FUNCTION "Generador de Fallas" : VOID	// FC 6
VERSION : 0.1
BEGIN
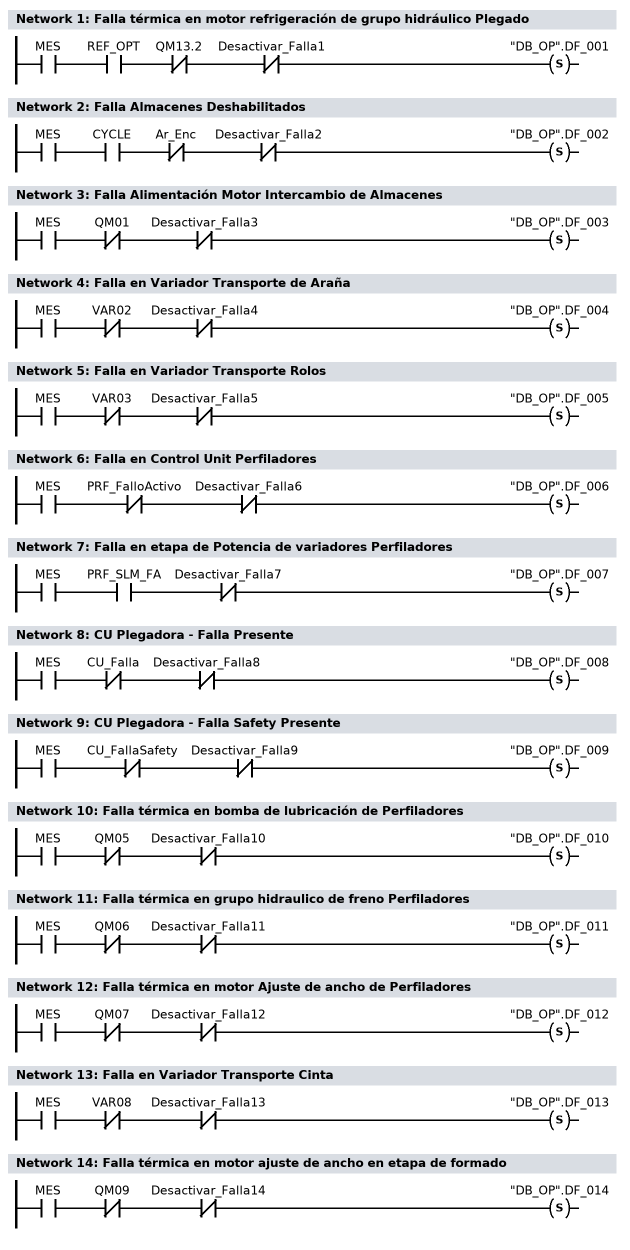
NETWORK
TITLE = Falla térmica en motor refrigeración de grupo hidráulico Plegado
      A     "MES";
      A     "REF_OPT";
      AN    "QM13.2";
      AN    "Desactivar_Falla1";
      S     "DB_OP".DF_001;
NETWORK
TITLE = Falla Almacenes Deshabilitados
      A     "MES";
      A     "CYCLE";
      AN    "Ar_Enc";
      AN    "Desactivar_Falla2";
      S     "DB_OP".DF_002;
NETWORK
TITLE = Falla Alimentación Motor Intercambio de Almacenes
      A     "MES";
      AN    "QM01";
      AN    "Desactivar_Falla3";
      S     "DB_OP".DF_003;
NETWORK
TITLE = Falla en Variador Transporte de Araña
      A     "MES";
      AN    "VAR02";
      AN    "Desactivar_Falla4";
      S     "DB_OP".DF_004;
NETWORK
TITLE = Falla en Variador Transporte Rolos
      A     "MES";
      AN    "VAR03";
      AN    "Desactivar_Falla5";
      S     "DB_OP".DF_005;
NETWORK
TITLE = Falla en Control Unit Perfiladores
      A     "MES";
      AN    "PRF_FalloActivo";
      AN    "Desactivar_Falla6";
      S     "DB_OP".DF_006;
NETWORK
TITLE = Falla en etapa de Potencia de variadores Perfiladores
      A     "MES";
      A     "PRF_SLM_FA";
      AN    "Desactivar_Falla7";
      S     "DB_OP".DF_007;
NETWORK
TITLE = CU Plegadora - Falla Presente
      A     "MES";
      AN    "CU_Falla";
      AN    "Desactivar_Falla8";
      S     "DB_OP".DF_008;
NETWORK
TITLE = CU Plegadora - Falla Safety Presente
      A     "MES";
      AN    "CU_FallaSafety";
      AN    "Desactivar_Falla9";
      S     "DB_OP".DF_009;
NETWORK
TITLE = Falla térmica en bomba de lubricación de Perfiladores
      A     "MES";
      AN    "QM05";
      AN    "Desactivar_Falla10";
      S     "DB_OP".DF_010;
NETWORK
TITLE = Falla térmica en grupo hidraulico de freno Perfiladores
      A     "MES";
      AN    "QM06";
      AN    "Desactivar_Falla11";
      S     "DB_OP".DF_011;
NETWORK
TITLE = Falla térmica en motor Ajuste de ancho de Perfiladores
      A     "MES";
      AN    "QM07";
      AN    "Desactivar_Falla12";
      S     "DB_OP".DF_012;
NETWORK
TITLE = Falla en Variador Transporte Cinta
      A     "MES";
      AN    "VAR08";
      AN    "Desactivar_Falla13";
      S     "DB_OP".DF_013;
NETWORK
TITLE = Falla térmica en motor ajuste de ancho en etapa de formado
      A     "MES";
      AN    "QM09";
      AN    "Desactivar_Falla14";
      S     "DB_OP".DF_014;
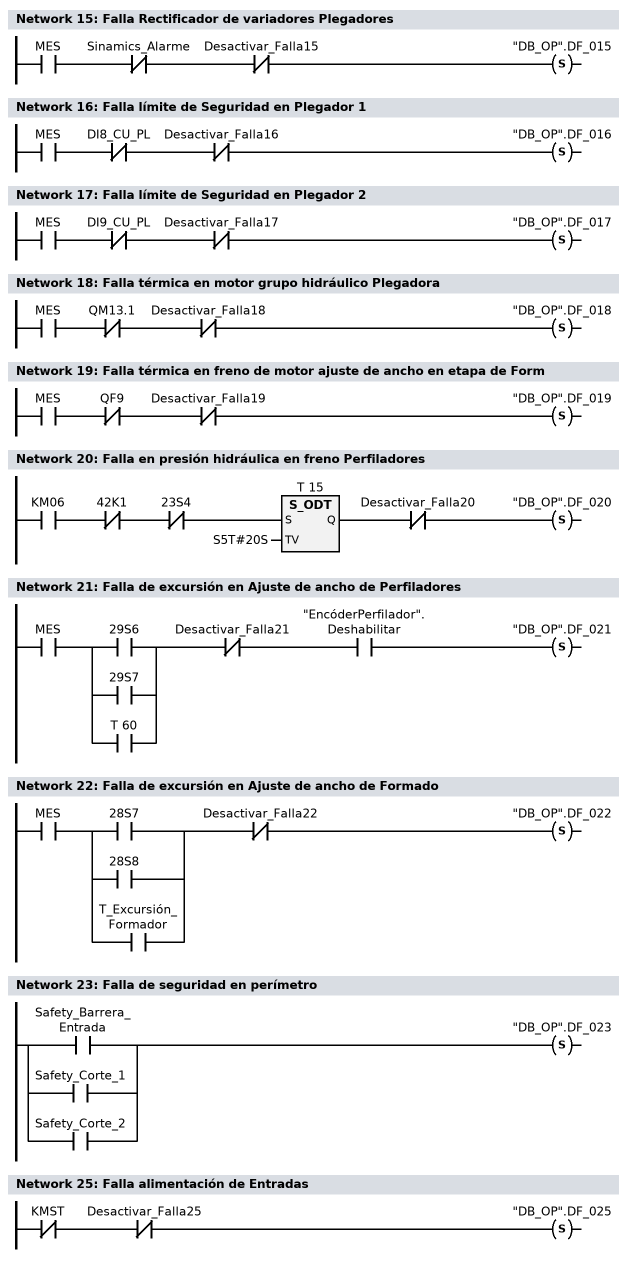
NETWORK
TITLE = Falla Rectificador de variadores Plegadores
      A     "MES";
      AN    "Sinamics_Alarme";
      AN    "Desactivar_Falla15";
      S     "DB_OP".DF_015;
NETWORK
TITLE = Falla límite de Seguridad en Plegador 1
      A     "MES";
      AN    "DI8_CU_PL";
      AN    "Desactivar_Falla16";
      S     "DB_OP".DF_016;
NETWORK
TITLE = Falla límite de Seguridad en Plegador 2
      A     "MES";
      AN    "DI9_CU_PL";
      AN    "Desactivar_Falla17";
      S     "DB_OP".DF_017;
NETWORK
TITLE = Falla térmica en motor grupo hidráulico Plegadora
      A     "MES";
      AN    "QM13.1";
      AN    "Desactivar_Falla18";
      S     "DB_OP".DF_018;
NETWORK
TITLE = Falla térmica en freno de motor ajuste de ancho en etapa de Form
      A     "MES";
      AN    "QF9";
      AN    "Desactivar_Falla19";
      S     "DB_OP".DF_019;
NETWORK
TITLE = Falla en presión hidráulica en freno Perfiladores
      A(;
      A     "KM06";
      AN    "42K1";
      AN    "23S4";
      L     S5T#20S;
      SD    T 15;
      NOP   0;
      NOP   0;
      NOP   0;
      A     T 15;
      );
      AN    "Desactivar_Falla20";
      S     "DB_OP".DF_020;
NETWORK
TITLE = Falla de excursión en Ajuste de ancho de Perfiladores
      A     "MES";
      A(;
      O     "29S6";
      O     "29S7";
      O     T 60;
      );
      AN    "Desactivar_Falla21";
      A     "EncóderPerfilador".Deshabilitar;
      S     "DB_OP".DF_021;
NETWORK
TITLE = Falla de excursión en Ajuste de ancho de Formado
      A     "MES";
      A(;
      O     "28S7";
      O     "28S8";
      O     "T_Excursión_Formador";
      );
      AN    "Desactivar_Falla22";
      S     "DB_OP".DF_022;
NETWORK
TITLE = Falla de seguridad en perímetro
      O     "Safety_Barrera_Entrada";
      O     "Safety_Corte_1";
      O     "Safety_Corte_2";
      S     "DB_OP".DF_023;
NETWORK
TITLE = Reserva
NETWORK
TITLE = Falla alimentación de Entradas
      AN    "KMST";
      AN    "Desactivar_Falla25";
      S     "DB_OP".DF_025;
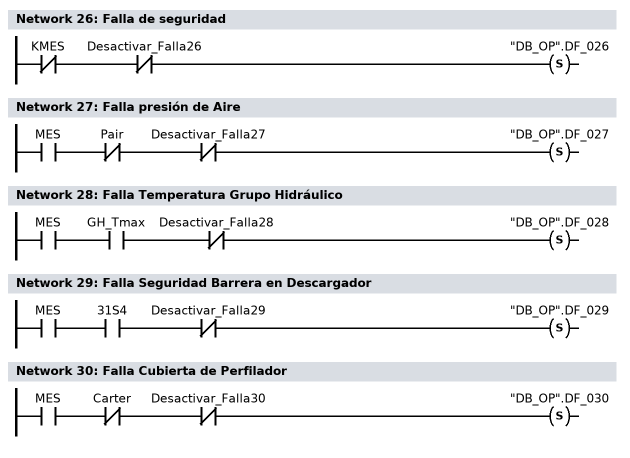
NETWORK
TITLE = Falla de seguridad
      AN    "KMES";
      AN    "Desactivar_Falla26";
      S     "DB_OP".DF_026;
NETWORK
TITLE = Falla presión de Aire
      A     "MES";
      AN    "Pair";
      AN    "Desactivar_Falla27";
      S     "DB_OP".DF_027;
NETWORK
TITLE = Falla Temperatura Grupo Hidráulico
      A     "MES";
      A     "GH_Tmax";
      AN    "Desactivar_Falla28";
      S     "DB_OP".DF_028;
NETWORK
TITLE = Falla Seguridad Barrera en Descargador
      A     "MES";
      A     "31S4";
      AN    "Desactivar_Falla29";
      S     "DB_OP".DF_029;
NETWORK
TITLE = Falla Cubierta de Perfilador
      A     "MES";
      AN    "Carter";
      AN    "Desactivar_Falla30";
      S     "DB_OP".DF_030;
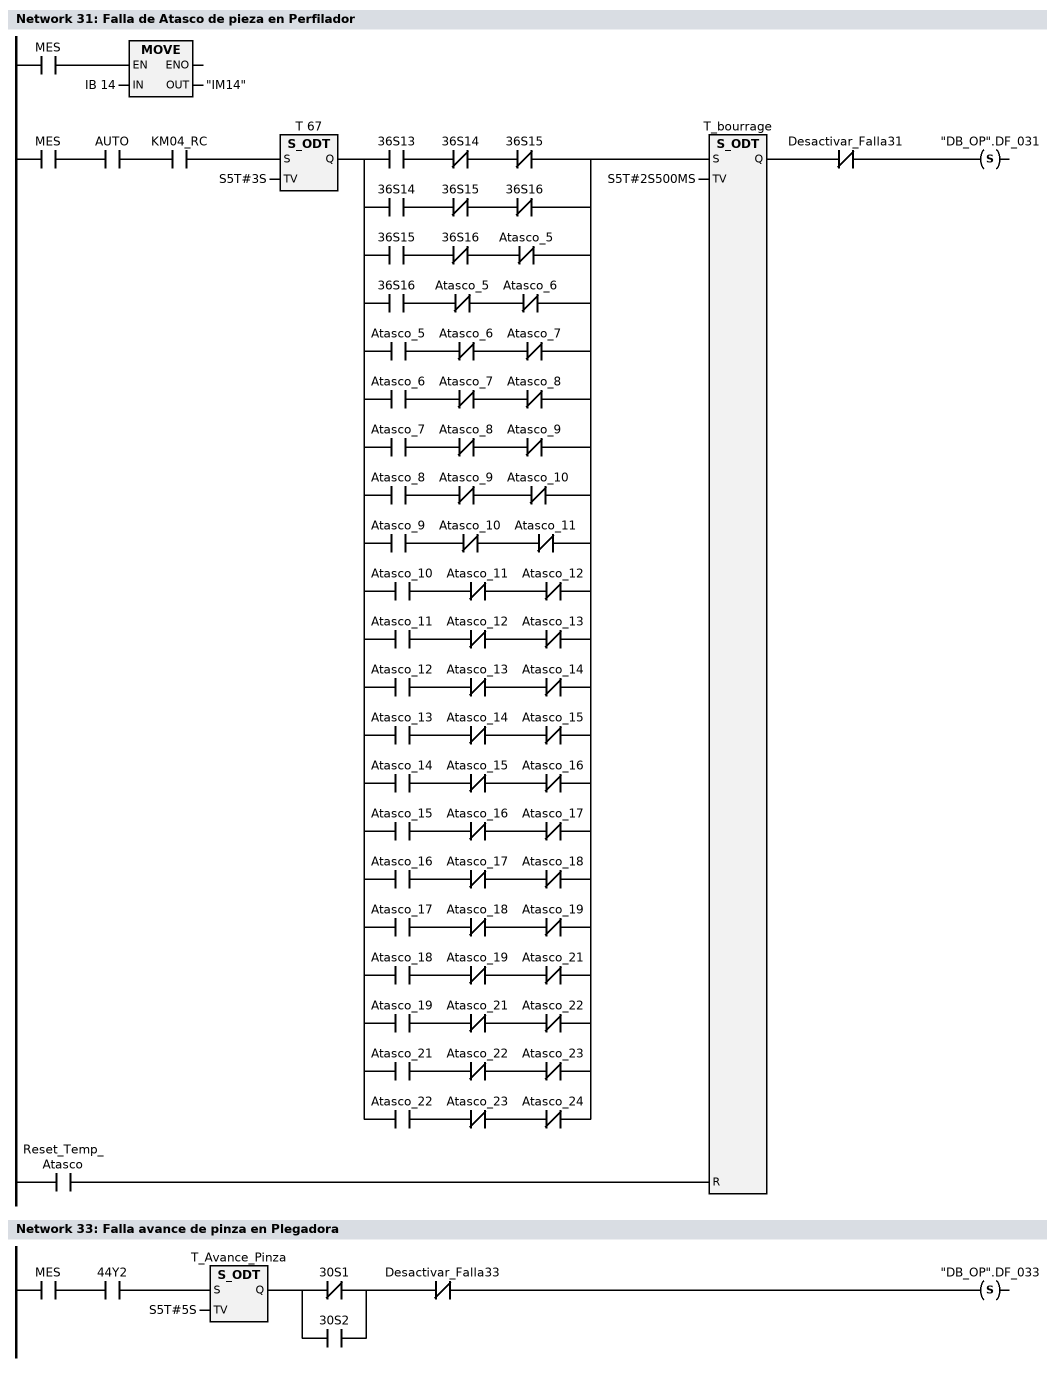
NETWORK
TITLE = Falla de Atasco de pieza en Perfilador
      A     "MES";
      =     L 0.0;
      A(;
      A(;
      A     L 0.0;
      A     "AUTO";
      A     "KM04_RC";
      L     S5T#3S;
      SD    T 67;
      NOP   0;
      NOP   0;
      NOP   0;
      A     T 67;
      );
      A(;
      A     "36S13";
      AN    "36S14";
      AN    "36S15";
      O;
      A     "36S14";
      AN    "36S15";
      AN    "36S16";
      O;
      A     "36S15";
      AN    "36S16";
      AN    "Atasco_5";
      O;
      A     "36S16";
      AN    "Atasco_5";
      AN    "Atasco_6";
      O;
      A     "Atasco_5";
      AN    "Atasco_6";
      AN    "Atasco_7";
      O;
      A     "Atasco_6";
      AN    "Atasco_7";
      AN    "Atasco_8";
      O;
      A     "Atasco_7";
      AN    "Atasco_8";
      AN    "Atasco_9";
      O;
      A     "Atasco_8";
      AN    "Atasco_9";
      AN    "Atasco_10";
      O;
      A     "Atasco_9";
      AN    "Atasco_10";
      AN    "Atasco_11";
      O;
      A     "Atasco_10";
      AN    "Atasco_11";
      AN    "Atasco_12";
      O;
      A     "Atasco_11";
      AN    "Atasco_12";
      AN    "Atasco_13";
      O;
      A     "Atasco_12";
      AN    "Atasco_13";
      AN    "Atasco_14";
      O;
      A     "Atasco_13";
      AN    "Atasco_14";
      AN    "Atasco_15";
      O;
      A     "Atasco_14";
      AN    "Atasco_15";
      AN    "Atasco_16";
      O;
      A     "Atasco_15";
      AN    "Atasco_16";
      AN    "Atasco_17";
      O;
      A     "Atasco_16";
      AN    "Atasco_17";
      AN    "Atasco_18";
      O;
      A     "Atasco_17";
      AN    "Atasco_18";
      AN    "Atasco_19";
      O;
      A     "Atasco_18";
      AN    "Atasco_19";
      AN    "Atasco_21";
      O;
      A     "Atasco_19";
      AN    "Atasco_21";
      AN    "Atasco_22";
      O;
      A     "Atasco_21";
      AN    "Atasco_22";
      AN    "Atasco_23";
      O;
      A     "Atasco_22";
      AN    "Atasco_23";
      AN    "Atasco_24";
      );
      L     S5T#2S500MS;
      SD    "T_bourrage";
      A     "Reset_Temp_Atasco";
      R     "T_bourrage";
      NOP   0;
      NOP   0;
      A     "T_bourrage";
      );
      AN    "Desactivar_Falla31";
      S     "DB_OP".DF_031;
      A     L 0.0;
      JNB   _001;
      L     IB 14;
      T     "IM14";
_001: NOP   0;
NETWORK
TITLE = Reserva
NETWORK
TITLE = Falla avance de pinza en Plegadora
      A(;
      A     "MES";
      A     "44Y2";
      L     S5T#5S;
      SD    "T_Avance_Pinza";
      NOP   0;
      NOP   0;
      NOP   0;
      A     "T_Avance_Pinza";
      );
      A(;
      ON    "30S1";
      O     "30S2";
      );
      AN    "Desactivar_Falla33";
      S     "DB_OP".DF_033;
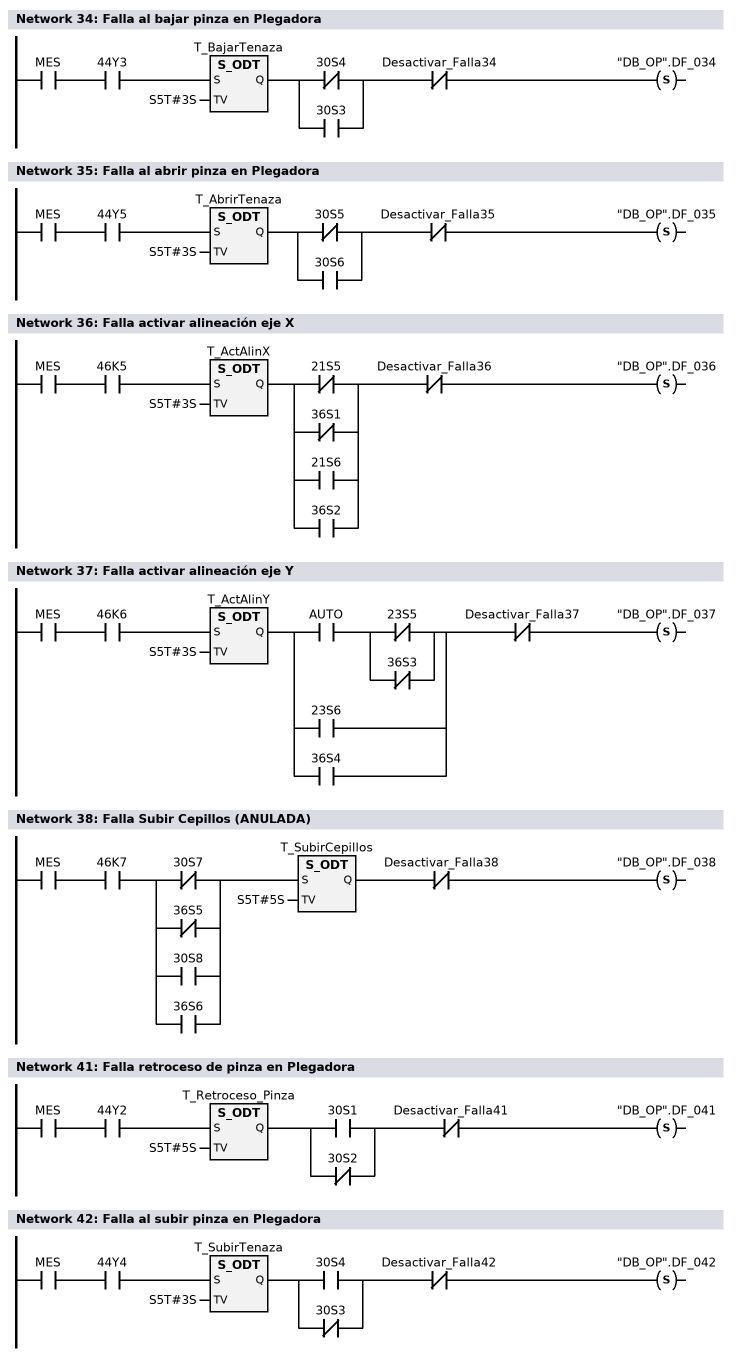
NETWORK
TITLE = Falla al bajar pinza en Plegadora
      A(;
      A     "MES";
      A     "44Y3";
      L     S5T#3S;
      SD    "T_BajarTenaza";
      NOP   0;
      NOP   0;
      NOP   0;
      A     "T_BajarTenaza";
      );
      A(;
      ON    "30S4";
      O     "30S3";
      );
      AN    "Desactivar_Falla34";
      S     "DB_OP".DF_034;
NETWORK
TITLE = Falla al abrir pinza en Plegadora
      A(;
      A     "MES";
      A     "44Y5";
      L     S5T#3S;
      SD    "T_AbrirTenaza";
      NOP   0;
      NOP   0;
      NOP   0;
      A     "T_AbrirTenaza";
      );
      A(;
      ON    "30S5";
      O     "30S6";
      );
      AN    "Desactivar_Falla35";
      S     "DB_OP".DF_035;
NETWORK
TITLE = Falla activar alineación eje X 
      A(;
      A     "MES";
      A     "46K5";
      L     S5T#3S;
      SD    "T_ActAlinX";
      NOP   0;
      NOP   0;
      NOP   0;
      A     "T_ActAlinX";
      );
      A(;
      ON    "21S5";
      ON    "36S1";
      O     "21S6";
      O     "36S2";
      );
      AN    "Desactivar_Falla36";
      S     "DB_OP".DF_036;
NETWORK
TITLE = Falla activar alineación eje Y 
      A(;
      A     "MES";
      A     "46K6";
      L     S5T#3S;
      SD    "T_ActAlinY";
      NOP   0;
      NOP   0;
      NOP   0;
      A     "T_ActAlinY";
      );
      A(;
      A     "AUTO";
      A(;
      ON    "23S5";
      ON    "36S3";
      );
      O     "23S6";
      O     "36S4";
      );
      AN    "Desactivar_Falla37";
      S     "DB_OP".DF_037;
NETWORK
TITLE = Falla Subir Cepillos (ANULADA)
      A(;
      A     "MES";
      A     "46K7";
      A(;
      ON    "30S7";
      ON    "36S5";
      O     "30S8";
      O     "36S6";
      );
      L     S5T#5S;
      SD    "T_SubirCepillos";
      NOP   0;
      NOP   0;
      NOP   0;
      A     "T_SubirCepillos";
      );
      AN    "Desactivar_Falla38";
      S     "DB_OP".DF_038;
NETWORK
TITLE = Reserva
NETWORK
TITLE = Reserva
NETWORK
TITLE = Falla retroceso de pinza en Plegadora
      A(;
      A     "MES";
      A     "44Y2";
      L     S5T#5S;
      SD    "T_Retroceso_Pinza";
      NOP   0;
      NOP   0;
      NOP   0;
      A     "T_Retroceso_Pinza";
      );
      A(;
      O     "30S1";
      ON    "30S2";
      );
      AN    "Desactivar_Falla41";
      S     "DB_OP".DF_041;
NETWORK
TITLE = Falla al subir pinza en Plegadora
      A(;
      A     "MES";
      A     "44Y4";
      L     S5T#3S;
      SD    "T_SubirTenaza";
      NOP   0;
      NOP   0;
      NOP   0;
      A     "T_SubirTenaza";
      );
      A(;
      O     "30S4";
      ON    "30S3";
      );
      AN    "Desactivar_Falla42";
      S     "DB_OP".DF_042;
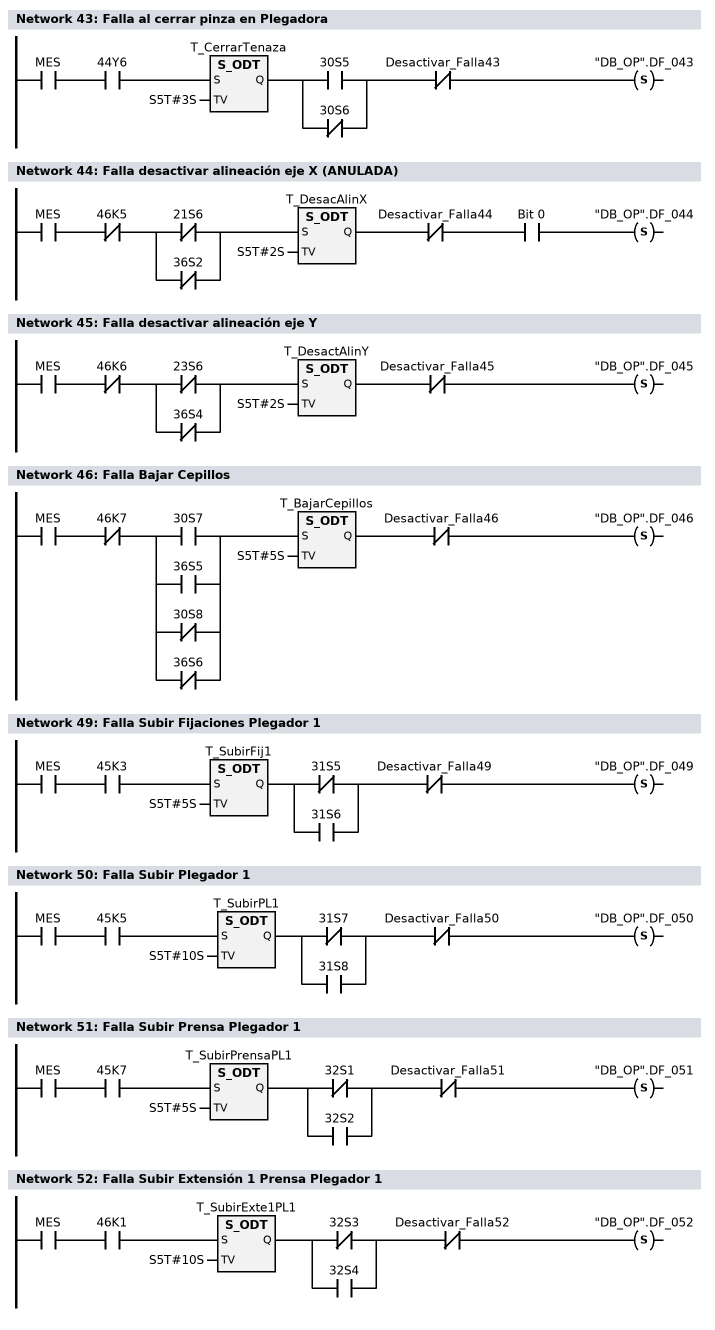
NETWORK
TITLE = Falla al cerrar pinza en Plegadora
      A(;
      A     "MES";
      A     "44Y6";
      L     S5T#3S;
      SD    "T_CerrarTenaza";
      NOP   0;
      NOP   0;
      NOP   0;
      A     "T_CerrarTenaza";
      );
      A(;
      O     "30S5";
      ON    "30S6";
      );
      AN    "Desactivar_Falla43";
      S     "DB_OP".DF_043;
NETWORK
TITLE = Falla desactivar alineación eje X (ANULADA)
      A(;
      A     "MES";
      AN    "46K5";
      A(;
      ON    "21S6";
      ON    "36S2";
      );
      L     S5T#2S;
      SD    "T_DesacAlinX";
      NOP   0;
      NOP   0;
      NOP   0;
      A     "T_DesacAlinX";
      );
      AN    "Desactivar_Falla44";
      A     "Bit 0";
      S     "DB_OP".DF_044;
NETWORK
TITLE = Falla desactivar alineación eje Y
      A(;
      A     "MES";
      AN    "46K6";
      A(;
      ON    "23S6";
      ON    "36S4";
      );
      L     S5T#2S;
      SD    "T_DesactAlinY";
      NOP   0;
      NOP   0;
      NOP   0;
      A     "T_DesactAlinY";
      );
      AN    "Desactivar_Falla45";
      S     "DB_OP".DF_045;
NETWORK
TITLE = Falla Bajar Cepillos 
      A(;
      A     "MES";
      AN    "46K7";
      A(;
      O     "30S7";
      O     "36S5";
      ON    "30S8";
      ON    "36S6";
      );
      L     S5T#5S;
      SD    "T_BajarCepillos";
      NOP   0;
      NOP   0;
      NOP   0;
      A     "T_BajarCepillos";
      );
      AN    "Desactivar_Falla46";
      S     "DB_OP".DF_046;
NETWORK
TITLE = Reserva
NETWORK
TITLE = Reserva
NETWORK
TITLE = Falla Subir Fijaciones Plegador 1
      A(;
      A     "MES";
      A     "45K3";
      L     S5T#5S;
      SD    "T_SubirFij1";
      NOP   0;
      NOP   0;
      NOP   0;
      A     "T_SubirFij1";
      );
      A(;
      ON    "31S5";
      O     "31S6";
      );
      AN    "Desactivar_Falla49";
      S     "DB_OP".DF_049;
NETWORK
TITLE = Falla Subir Plegador 1
      A(;
      A     "MES";
      A     "45K5";
      L     S5T#10S;
      SD    "T_SubirPL1";
      NOP   0;
      NOP   0;
      NOP   0;
      A     "T_SubirPL1";
      );
      A(;
      ON    "31S7";
      O     "31S8";
      );
      AN    "Desactivar_Falla50";
      S     "DB_OP".DF_050;
NETWORK
TITLE = Falla Subir Prensa Plegador 1
      A(;
      A     "MES";
      A     "45K7";
      L     S5T#5S;
      SD    "T_SubirPrensaPL1";
      NOP   0;
      NOP   0;
      NOP   0;
      A     "T_SubirPrensaPL1";
      );
      A(;
      ON    "32S1";
      O     "32S2";
      );
      AN    "Desactivar_Falla51";
      S     "DB_OP".DF_051;
NETWORK
TITLE = Falla Subir Extensión 1 Prensa Plegador 1
      A(;
      A     "MES";
      A     "46K1";
      L     S5T#10S;
      SD    "T_SubirExte1PL1";
      NOP   0;
      NOP   0;
      NOP   0;
      A     "T_SubirExte1PL1";
      );
      A(;
      ON    "32S3";
      O     "32S4";
      );
      AN    "Desactivar_Falla52";
      S     "DB_OP".DF_052;
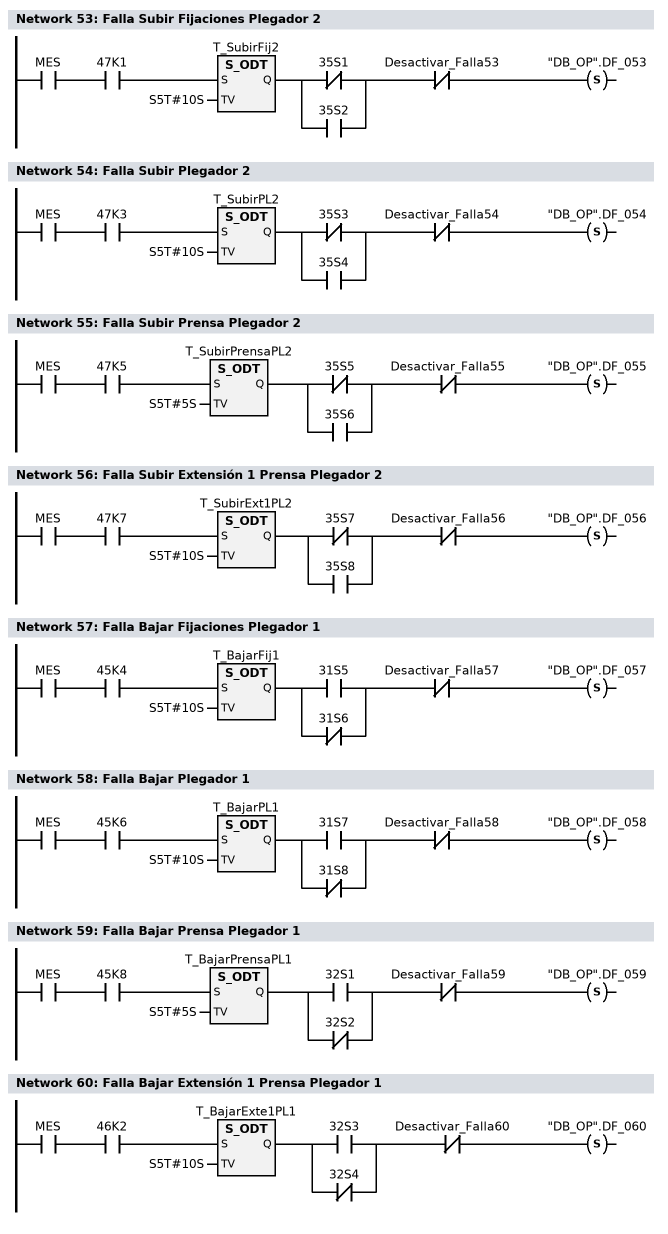
NETWORK
TITLE = Falla Subir Fijaciones Plegador 2
      A(;
      A     "MES";
      A     "47K1";
      L     S5T#10S;
      SD    "T_SubirFij2";
      NOP   0;
      NOP   0;
      NOP   0;
      A     "T_SubirFij2";
      );
      A(;
      ON    "35S1";
      O     "35S2";
      );
      AN    "Desactivar_Falla53";
      S     "DB_OP".DF_053;
NETWORK
TITLE = Falla Subir Plegador 2
      A(;
      A     "MES";
      A     "47K3";
      L     S5T#10S;
      SD    "T_SubirPL2";
      NOP   0;
      NOP   0;
      NOP   0;
      A     "T_SubirPL2";
      );
      A(;
      ON    "35S3";
      O     "35S4";
      );
      AN    "Desactivar_Falla54";
      S     "DB_OP".DF_054;
NETWORK
TITLE = Falla Subir Prensa Plegador 2
      A(;
      A     "MES";
      A     "47K5";
      L     S5T#5S;
      SD    "T_SubirPrensaPL2";
      NOP   0;
      NOP   0;
      NOP   0;
      A     "T_SubirPrensaPL2";
      );
      A(;
      ON    "35S5";
      O     "35S6";
      );
      AN    "Desactivar_Falla55";
      S     "DB_OP".DF_055;
NETWORK
TITLE = Falla Subir Extensión 1 Prensa Plegador 2
      A(;
      A     "MES";
      A     "47K7";
      L     S5T#10S;
      SD    "T_SubirExt1PL2";
      NOP   0;
      NOP   0;
      NOP   0;
      A     "T_SubirExt1PL2";
      );
      A(;
      ON    "35S7";
      O     "35S8";
      );
      AN    "Desactivar_Falla56";
      S     "DB_OP".DF_056;
NETWORK
TITLE = Falla Bajar Fijaciones Plegador 1
      A(;
      A     "MES";
      A     "45K4";
      L     S5T#10S;
      SD    "T_BajarFij1";
      NOP   0;
      NOP   0;
      NOP   0;
      A     "T_BajarFij1";
      );
      A(;
      O     "31S5";
      ON    "31S6";
      );
      AN    "Desactivar_Falla57";
      S     "DB_OP".DF_057;
NETWORK
TITLE = Falla Bajar Plegador 1
      A(;
      A     "MES";
      A     "45K6";
      L     S5T#10S;
      SD    "T_BajarPL1";
      NOP   0;
      NOP   0;
      NOP   0;
      A     "T_BajarPL1";
      );
      A(;
      O     "31S7";
      ON    "31S8";
      );
      AN    "Desactivar_Falla58";
      S     "DB_OP".DF_058;
NETWORK
TITLE = Falla Bajar Prensa Plegador 1
      A(;
      A     "MES";
      A     "45K8";
      L     S5T#5S;
      SD    "T_BajarPrensaPL1";
      NOP   0;
      NOP   0;
      NOP   0;
      A     "T_BajarPrensaPL1";
      );
      A(;
      O     "32S1";
      ON    "32S2";
      );
      AN    "Desactivar_Falla59";
      S     "DB_OP".DF_059;
NETWORK
TITLE = Falla Bajar Extensión 1 Prensa Plegador 1
      A(;
      A     "MES";
      A     "46K2";
      L     S5T#10S;
      SD    "T_BajarExte1PL1";
      NOP   0;
      NOP   0;
      NOP   0;
      A     "T_BajarExte1PL1";
      );
      A(;
      O     "32S3";
      ON    "32S4";
      );
      AN    "Desactivar_Falla60";
      S     "DB_OP".DF_060;
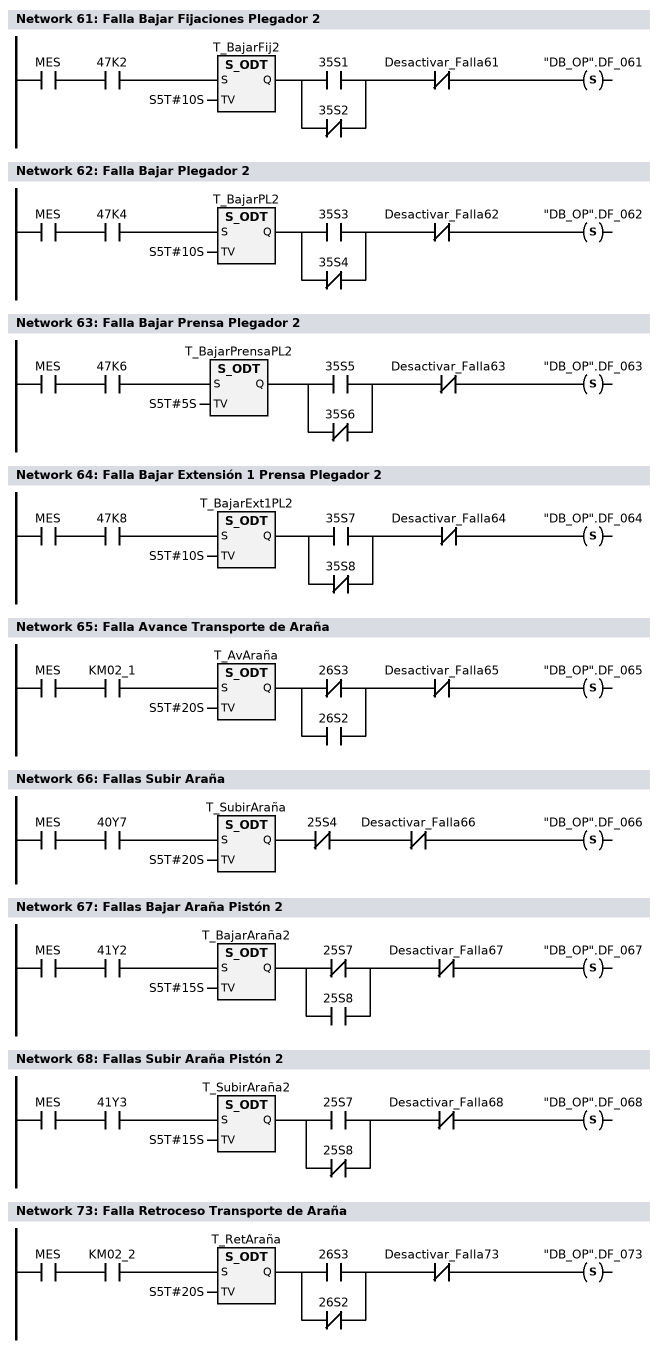
NETWORK
TITLE = Falla Bajar Fijaciones Plegador 2
      A(;
      A     "MES";
      A     "47K2";
      L     S5T#10S;
      SD    "T_BajarFij2";
      NOP   0;
      NOP   0;
      NOP   0;
      A     "T_BajarFij2";
      );
      A(;
      O     "35S1";
      ON    "35S2";
      );
      AN    "Desactivar_Falla61";
      S     "DB_OP".DF_061;
NETWORK
TITLE = Falla Bajar Plegador 2
      A(;
      A     "MES";
      A     "47K4";
      L     S5T#10S;
      SD    "T_BajarPL2";
      NOP   0;
      NOP   0;
      NOP   0;
      A     "T_BajarPL2";
      );
      A(;
      O     "35S3";
      ON    "35S4";
      );
      AN    "Desactivar_Falla62";
      S     "DB_OP".DF_062;
NETWORK
TITLE = Falla Bajar Prensa Plegador 2
      A(;
      A     "MES";
      A     "47K6";
      L     S5T#5S;
      SD    "T_BajarPrensaPL2";
      NOP   0;
      NOP   0;
      NOP   0;
      A     "T_BajarPrensaPL2";
      );
      A(;
      O     "35S5";
      ON    "35S6";
      );
      AN    "Desactivar_Falla63";
      S     "DB_OP".DF_063;
NETWORK
TITLE = Falla Bajar Extensión 1 Prensa Plegador 2
      A(;
      A     "MES";
      A     "47K8";
      L     S5T#10S;
      SD    "T_BajarExt1PL2";
      NOP   0;
      NOP   0;
      NOP   0;
      A     "T_BajarExt1PL2";
      );
      A(;
      O     "35S7";
      ON    "35S8";
      );
      AN    "Desactivar_Falla64";
      S     "DB_OP".DF_064;
NETWORK
TITLE = Falla Avance Transporte de Araña
      A(;
      A     "MES";
      A     "KM02_1";
      L     S5T#20S;
      SD    "T_AvAraña";
      NOP   0;
      NOP   0;
      NOP   0;
      A     "T_AvAraña";
      );
      A(;
      ON    "26S3";
      O     "26S2";
      );
      AN    "Desactivar_Falla65";
      S     "DB_OP".DF_065;
NETWORK
TITLE = Fallas Subir Araña
      A(;
      A     "MES";
      A     "40Y7";
      L     S5T#20S;
      SD    "T_SubirAraña";
      NOP   0;
      NOP   0;
      NOP   0;
      A     "T_SubirAraña";
      );
      AN    "25S4";
      AN    "Desactivar_Falla66";
      S     "DB_OP".DF_066;
NETWORK
TITLE = Fallas Bajar Araña Pistón 2
      A(;
      A     "MES";
      A     "41Y2";
      L     S5T#15S;
      SD    "T_BajarAraña2";
      NOP   0;
      NOP   0;
      NOP   0;
      A     "T_BajarAraña2";
      );
      A(;
      ON    "25S7";
      O     "25S8";
      );
      AN    "Desactivar_Falla67";
      S     "DB_OP".DF_067;
NETWORK
TITLE = Fallas Subir Araña Pistón 2
      A(;
      A     "MES";
      A     "41Y3";
      L     S5T#15S;
      SD    "T_SubirAraña2";
      NOP   0;
      NOP   0;
      NOP   0;
      A     "T_SubirAraña2";
      );
      A(;
      O     "25S7";
      ON    "25S8";
      );
      AN    "Desactivar_Falla68";
      S     "DB_OP".DF_068;
NETWORK
TITLE = Reserva
NETWORK
TITLE = Reserva
NETWORK
TITLE = Reserva
NETWORK
TITLE = Reserva
NETWORK
TITLE = Falla Retroceso Transporte de Araña
      A(;
      A     "MES";
      A     "KM02_2";
      L     S5T#20S;
      SD    "T_RetAraña";
      NOP   0;
      NOP   0;
      NOP   0;
      A     "T_RetAraña";
      );
      A(;
      O     "26S3";
      ON    "26S2";
      );
      AN    "Desactivar_Falla73";
      S     "DB_OP".DF_073;
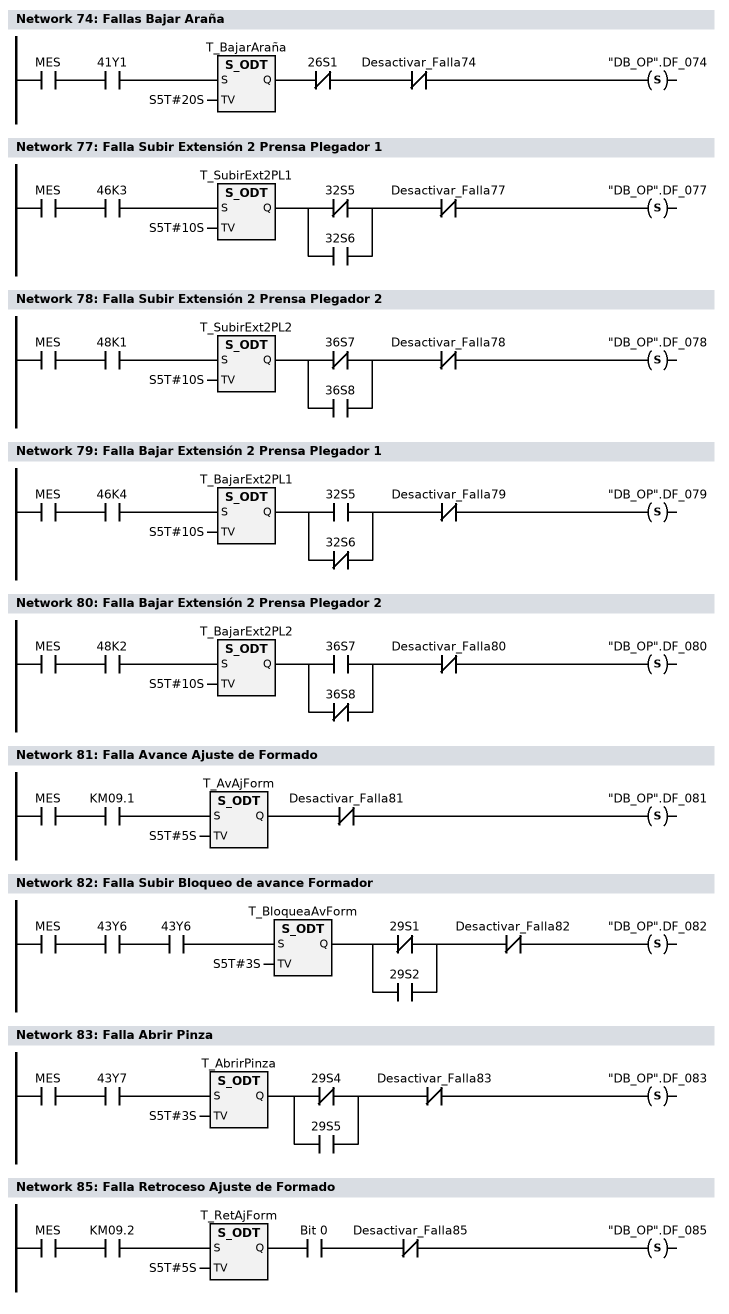
NETWORK
TITLE = Fallas Bajar Araña
      A(;
      A     "MES";
      A     "41Y1";
      L     S5T#20S;
      SD    "T_BajarAraña";
      NOP   0;
      NOP   0;
      NOP   0;
      A     "T_BajarAraña";
      );
      AN    "26S1";
      AN    "Desactivar_Falla74";
      S     "DB_OP".DF_074;
NETWORK
TITLE = Reserva
NETWORK
TITLE = Reserva
NETWORK
TITLE = Falla Subir Extensión 2 Prensa Plegador 1
      A(;
      A     "MES";
      A     "46K3";
      L     S5T#10S;
      SD    "T_SubirExt2PL1";
      NOP   0;
      NOP   0;
      NOP   0;
      A     "T_SubirExt2PL1";
      );
      A(;
      ON    "32S5";
      O     "32S6";
      );
      AN    "Desactivar_Falla77";
      S     "DB_OP".DF_077;
NETWORK
TITLE = Falla Subir Extensión 2 Prensa Plegador 2
      A(;
      A     "MES";
      A     "48K1";
      L     S5T#10S;
      SD    "T_SubirExt2PL2";
      NOP   0;
      NOP   0;
      NOP   0;
      A     "T_SubirExt2PL2";
      );
      A(;
      ON    "36S7";
      O     "36S8";
      );
      AN    "Desactivar_Falla78";
      S     "DB_OP".DF_078;
NETWORK
TITLE = Falla Bajar Extensión 2 Prensa Plegador 1
      A(;
      A     "MES";
      A     "46K4";
      L     S5T#10S;
      SD    "T_BajarExt2PL1";
      NOP   0;
      NOP   0;
      NOP   0;
      A     "T_BajarExt2PL1";
      );
      A(;
      O     "32S5";
      ON    "32S6";
      );
      AN    "Desactivar_Falla79";
      S     "DB_OP".DF_079;
NETWORK
TITLE = Falla Bajar Extensión 2 Prensa Plegador 2
      A(;
      A     "MES";
      A     "48K2";
      L     S5T#10S;
      SD    "T_BajarExt2PL2";
      NOP   0;
      NOP   0;
      NOP   0;
      A     "T_BajarExt2PL2";
      );
      A(;
      O     "36S7";
      ON    "36S8";
      );
      AN    "Desactivar_Falla80";
      S     "DB_OP".DF_080;
NETWORK
TITLE = Falla Avance Ajuste de Formado
      A(;
      A     "MES";
      A     "KM09.1";
      L     S5T#5S;
      SD    "T_AvAjForm";
      NOP   0;
      NOP   0;
      NOP   0;
      A     "T_AvAjForm";
      );
      AN    "Desactivar_Falla81";
      S     "DB_OP".DF_081;
NETWORK
TITLE = Falla Subir Bloqueo de avance Formador
      A(;
      A     "MES";
      A     "43Y6";
      A     "43Y6";
      L     S5T#3S;
      SD    "T_BloqueaAvForm";
      NOP   0;
      NOP   0;
      NOP   0;
      A     "T_BloqueaAvForm";
      );
      A(;
      ON    "29S1";
      O     "29S2";
      );
      AN    "Desactivar_Falla82";
      S     "DB_OP".DF_082;
NETWORK
TITLE = Falla Abrir Pinza
      A(;
      A     "MES";
      A     "43Y7";
      L     S5T#3S;
      SD    "T_AbrirPinza";
      NOP   0;
      NOP   0;
      NOP   0;
      A     "T_AbrirPinza";
      );
      A(;
      ON    "29S4";
      O     "29S5";
      );
      AN    "Desactivar_Falla83";
      S     "DB_OP".DF_083;
NETWORK
TITLE = Reserva
NETWORK
TITLE = Falla Retroceso Ajuste de Formado
      A(;
      A     "MES";
      A     "KM09.2";
      L     S5T#5S;
      SD    "T_RetAjForm";
      NOP   0;
      NOP   0;
      NOP   0;
      A     "T_RetAjForm";
      );
      A     "Bit 0";
      AN    "Desactivar_Falla85";
      S     "DB_OP".DF_085;
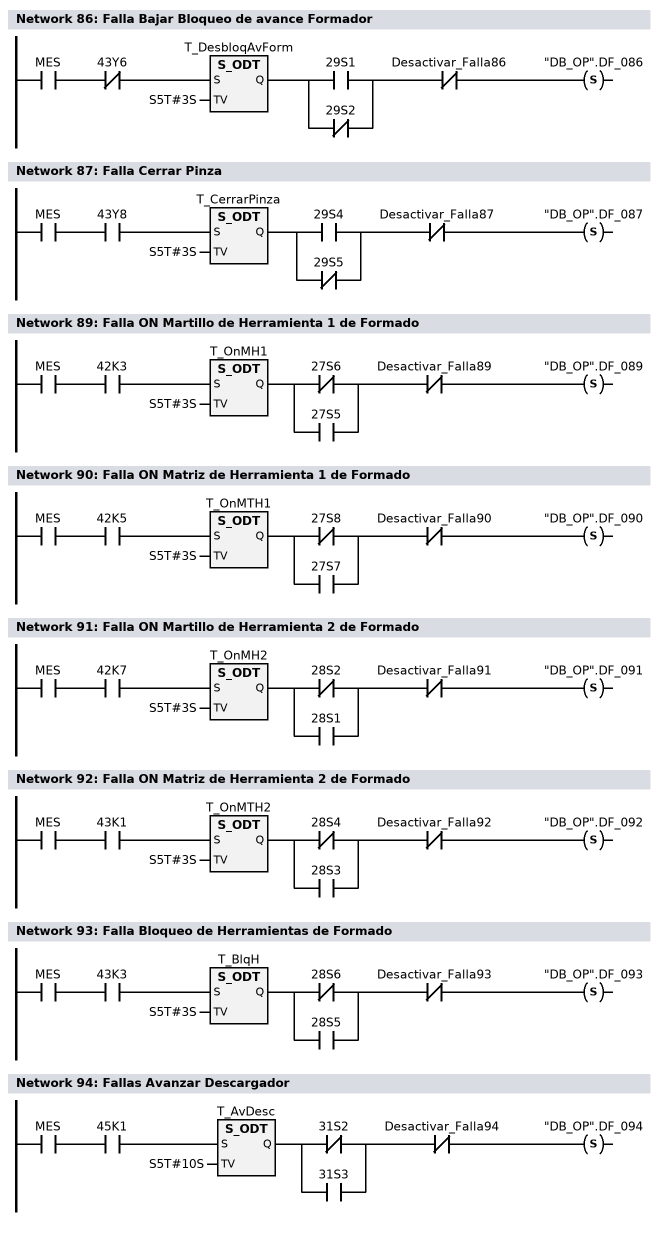
NETWORK
TITLE = Falla Bajar Bloqueo de avance Formador
      A(;
      A     "MES";
      AN    "43Y6";
      L     S5T#3S;
      SD    "T_DesbloqAvForm";
      NOP   0;
      NOP   0;
      NOP   0;
      A     "T_DesbloqAvForm";
      );
      A(;
      O     "29S1";
      ON    "29S2";
      );
      AN    "Desactivar_Falla86";
      S     "DB_OP".DF_086;
NETWORK
TITLE = Falla Cerrar Pinza
      A(;
      A     "MES";
      A     "43Y8";
      L     S5T#3S;
      SD    "T_CerrarPinza";
      NOP   0;
      NOP   0;
      NOP   0;
      A     "T_CerrarPinza";
      );
      A(;
      O     "29S4";
      ON    "29S5";
      );
      AN    "Desactivar_Falla87";
      S     "DB_OP".DF_087;
NETWORK
TITLE = Reserva
NETWORK
TITLE = Falla ON Martillo de Herramienta 1 de Formado 
      A(;
      A     "MES";
      A     "42K3";
      L     S5T#3S;
      SD    "T_OnMH1";
      NOP   0;
      NOP   0;
      NOP   0;
      A     "T_OnMH1";
      );
      A(;
      ON    "27S6";
      O     "27S5";
      );
      AN    "Desactivar_Falla89";
      S     "DB_OP".DF_089;
NETWORK
TITLE = Falla ON Matriz de Herramienta 1 de Formado 
      A(;
      A     "MES";
      A     "42K5";
      L     S5T#3S;
      SD    "T_OnMTH1";
      NOP   0;
      NOP   0;
      NOP   0;
      A     "T_OnMTH1";
      );
      A(;
      ON    "27S8";
      O     "27S7";
      );
      AN    "Desactivar_Falla90";
      S     "DB_OP".DF_090;
NETWORK
TITLE = Falla ON Martillo de Herramienta 2 de Formado
      A(;
      A     "MES";
      A     "42K7";
      L     S5T#3S;
      SD    "T_OnMH2";
      NOP   0;
      NOP   0;
      NOP   0;
      A     "T_OnMH2";
      );
      A(;
      ON    "28S2";
      O     "28S1";
      );
      AN    "Desactivar_Falla91";
      S     "DB_OP".DF_091;
NETWORK
TITLE = Falla ON Matriz de Herramienta 2 de Formado 
      A(;
      A     "MES";
      A     "43K1";
      L     S5T#3S;
      SD    "T_OnMTH2";
      NOP   0;
      NOP   0;
      NOP   0;
      A     "T_OnMTH2";
      );
      A(;
      ON    "28S4";
      O     "28S3";
      );
      AN    "Desactivar_Falla92";
      S     "DB_OP".DF_092;
NETWORK
TITLE = Falla Bloqueo de Herramientas de Formado 
      A(;
      A     "MES";
      A     "43K3";
      L     S5T#3S;
      SD    "T_BlqH";
      NOP   0;
      NOP   0;
      NOP   0;
      A     "T_BlqH";
      );
      A(;
      ON    "28S6";
      O     "28S5";
      );
      AN    "Desactivar_Falla93";
      S     "DB_OP".DF_093;
NETWORK
TITLE = Fallas Avanzar Descargador
      A(;
      A     "MES";
      A     "45K1";
      L     S5T#10S;
      SD    "T_AvDesc";
      NOP   0;
      NOP   0;
      NOP   0;
      A     "T_AvDesc";
      );
      A(;
      ON    "31S2";
      O     "31S3";
      );
      AN    "Desactivar_Falla94";
      S     "DB_OP".DF_094;
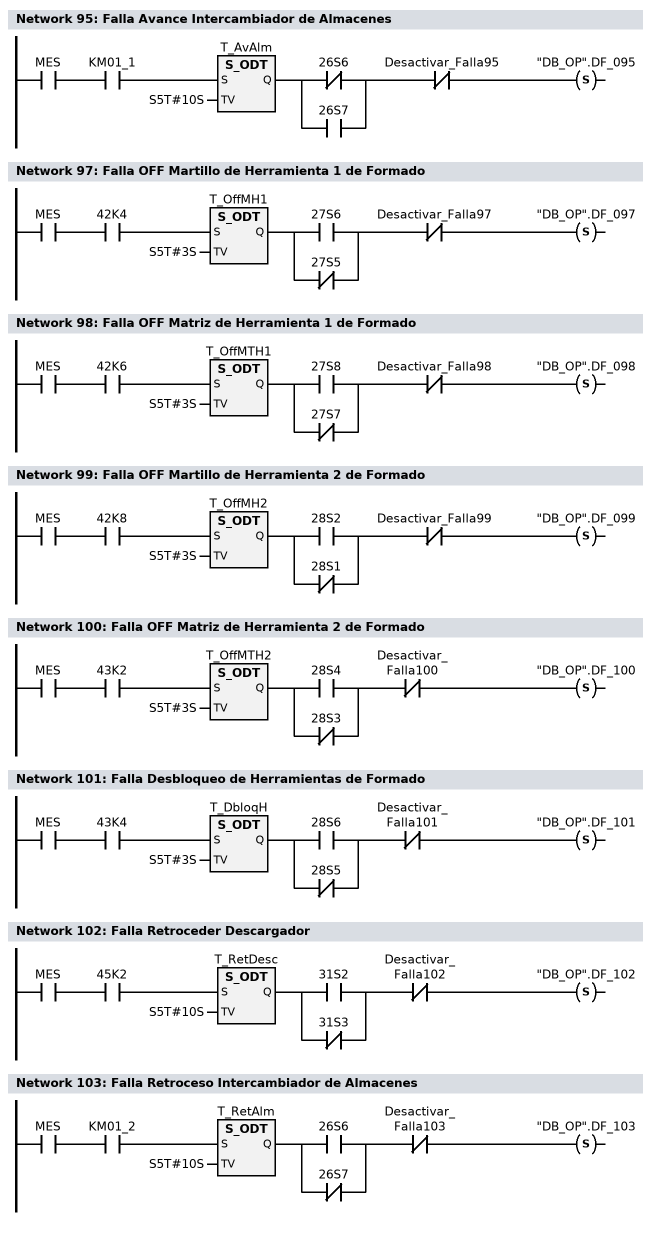
NETWORK
TITLE = Falla Avance Intercambiador de Almacenes
      A(;
      A     "MES";
      A     "KM01_1";
      L     S5T#10S;
      SD    "T_AvAlm";
      NOP   0;
      NOP   0;
      NOP   0;
      A     "T_AvAlm";
      );
      A(;
      ON    "26S6";
      O     "26S7";
      );
      AN    "Desactivar_Falla95";
      S     "DB_OP".DF_095;
NETWORK
TITLE = Reserva
NETWORK
TITLE = Falla OFF Martillo de Herramienta 1 de Formado 
      A(;
      A     "MES";
      A     "42K4";
      L     S5T#3S;
      SD    "T_OffMH1";
      NOP   0;
      NOP   0;
      NOP   0;
      A     "T_OffMH1";
      );
      A(;
      O     "27S6";
      ON    "27S5";
      );
      AN    "Desactivar_Falla97";
      S     "DB_OP".DF_097;
NETWORK
TITLE = Falla OFF Matriz de Herramienta 1 de Formado 
      A(;
      A     "MES";
      A     "42K6";
      L     S5T#3S;
      SD    "T_OffMTH1";
      NOP   0;
      NOP   0;
      NOP   0;
      A     "T_OffMTH1";
      );
      A(;
      O     "27S8";
      ON    "27S7";
      );
      AN    "Desactivar_Falla98";
      S     "DB_OP".DF_098;
NETWORK
TITLE = Falla OFF Martillo de Herramienta 2 de Formado
      A(;
      A     "MES";
      A     "42K8";
      L     S5T#3S;
      SD    "T_OffMH2";
      NOP   0;
      NOP   0;
      NOP   0;
      A     "T_OffMH2";
      );
      A(;
      O     "28S2";
      ON    "28S1";
      );
      AN    "Desactivar_Falla99";
      S     "DB_OP".DF_099;
NETWORK
TITLE = Falla OFF Matriz de Herramienta 2 de Formado 
      A(;
      A     "MES";
      A     "43K2";
      L     S5T#3S;
      SD    "T_OffMTH2";
      NOP   0;
      NOP   0;
      NOP   0;
      A     "T_OffMTH2";
      );
      A(;
      O     "28S4";
      ON    "28S3";
      );
      AN    "Desactivar_Falla100";
      S     "DB_OP".DF_100;
NETWORK
TITLE = Falla Desbloqueo de Herramientas de Formado 
      A(;
      A     "MES";
      A     "43K4";
      L     S5T#3S;
      SD    "T_DbloqH";
      NOP   0;
      NOP   0;
      NOP   0;
      A     "T_DbloqH";
      );
      A(;
      O     "28S6";
      ON    "28S5";
      );
      AN    "Desactivar_Falla101";
      S     "DB_OP".DF_101;
NETWORK
TITLE = Falla Retroceder Descargador
      A(;
      A     "MES";
      A     "45K2";
      L     S5T#10S;
      SD    "T_RetDesc";
      NOP   0;
      NOP   0;
      NOP   0;
      A     "T_RetDesc";
      );
      A(;
      O     "31S2";
      ON    "31S3";
      );
      AN    "Desactivar_Falla102";
      S     "DB_OP".DF_102;
NETWORK
TITLE = Falla Retroceso Intercambiador de Almacenes
      A(;
      A     "MES";
      A     "KM01_2";
      L     S5T#10S;
      SD    "T_RetAlm";
      NOP   0;
      NOP   0;
      NOP   0;
      A     "T_RetAlm";
      );
      A(;
      O     "26S6";
      ON    "26S7";
      );
      AN    "Desactivar_Falla103";
      S     "DB_OP".DF_103;
NETWORK
TITLE = Reserva
NETWORK
TITLE = Reserva
NETWORK
TITLE = Reserva
NETWORK
TITLE = Reserva
NETWORK
TITLE = Reserva
NETWORK
TITLE = Reserva
NETWORK
TITLE = Reserva
NETWORK
TITLE = Reserva
NETWORK
TITLE = Reserva
NETWORK
TITLE = Reserva
NETWORK
TITLE = Reserva
NETWORK
TITLE = Reserva
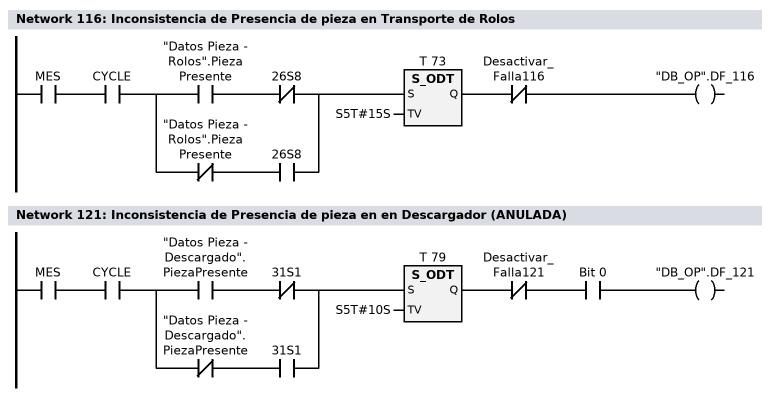
NETWORK
TITLE = Inconsistencia de Presencia de pieza en Transporte de Rolos
      A(;
      A     "MES";
      A     "CYCLE";
      A(;
      A     "Datos Pieza - Rolos".PiezaPresente;
      AN    "26S8";
      O;
      AN    "Datos Pieza - Rolos".PiezaPresente;
      A     "26S8";
      );
      L     S5T#15S;
      SD    T 73;
      NOP   0;
      NOP   0;
      NOP   0;
      A     T 73;
      );
      AN    "Desactivar_Falla116";
      =     "DB_OP".DF_116;
NETWORK
TITLE = Reserva
NETWORK
TITLE = Reserva
NETWORK
TITLE = Reserva
NETWORK
TITLE = Reserva
NETWORK
TITLE = Inconsistencia de Presencia de pieza en en Descargador (ANULADA)
      A(;
      A     "MES";
      A     "CYCLE";
      A(;
      A     "Datos Pieza - Descargado".PiezaPresente;
      AN    "31S1";
      O;
      AN    "Datos Pieza - Descargado".PiezaPresente;
      A     "31S1";
      );
      L     S5T#10S;
      SD    T 79;
      NOP   0;
      NOP   0;
      NOP   0;
      A     T 79;
      );
      AN    "Desactivar_Falla121";
      A     "Bit 0";
      =     "DB_OP".DF_121;
END_FUNCTION

FUNCTION "Asistencia" : VOID	// FC 8
AUTHOR : EMR
NAME : eProC
VERSION : 0.1
BEGIN
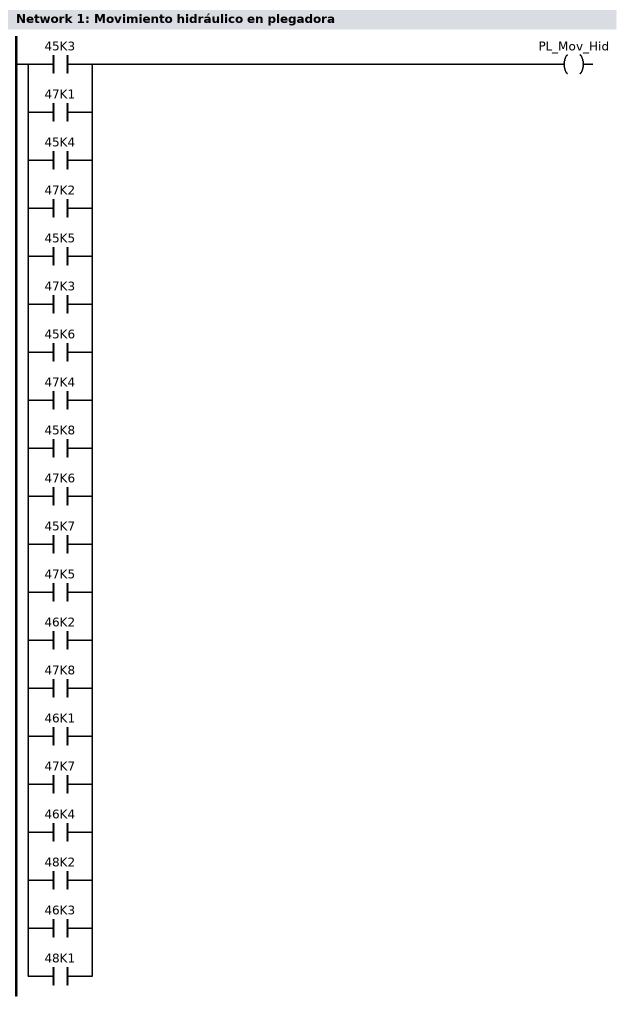
NETWORK
TITLE = Movimiento hidráulico en plegadora
      O     "45K3";
      O     "47K1";
      O     "45K4";
      O     "47K2";
      O     "45K5";
      O     "47K3";
      O     "45K6";
      O     "47K4";
      O     "45K8";
      O     "47K6";
      O     "45K7";
      O     "47K5";
      O     "46K2";
      O     "47K8";
      O     "46K1";
      O     "47K7";
      O     "46K4";
      O     "48K2";
      O     "46K3";
      O     "48K1";
      =     "PL_Mov_Hid";
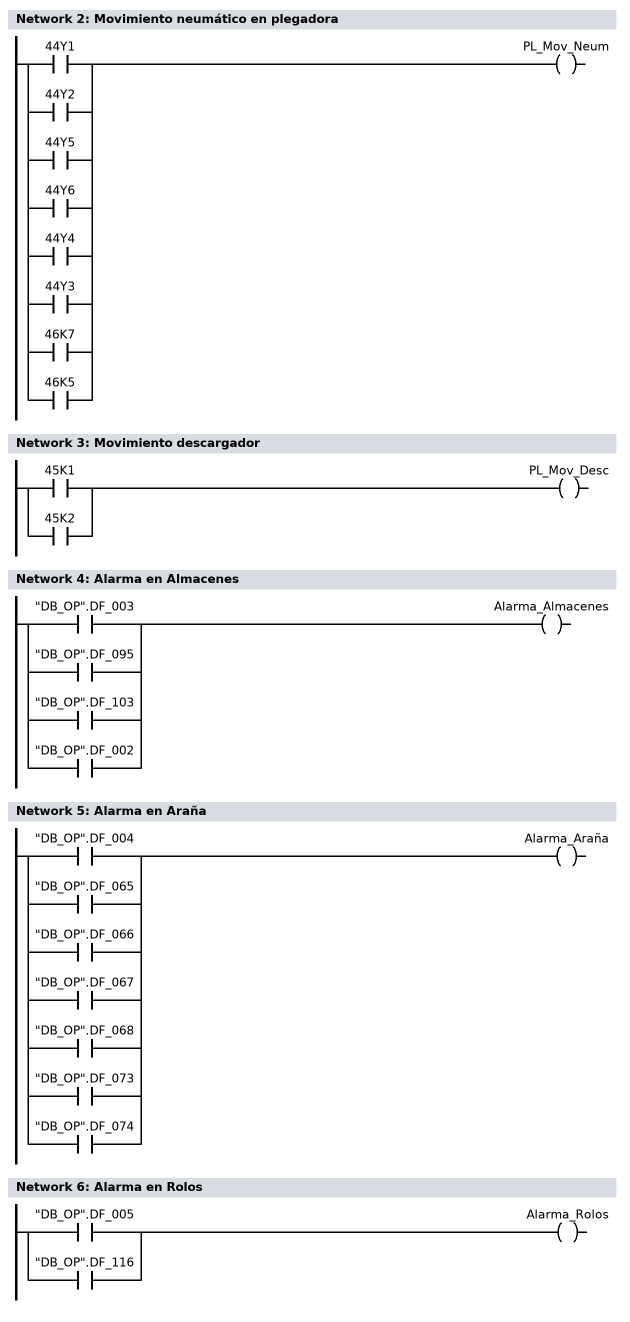
NETWORK
TITLE = Movimiento neumático en plegadora
      O     "44Y1";
      O     "44Y2";
      O     "44Y5";
      O     "44Y6";
      O     "44Y4";
      O     "44Y3";
      O     "46K7";
      O     "46K5";
      =     "PL_Mov_Neum";
NETWORK
TITLE = Movimiento descargador
      O     "45K1";
      O     "45K2";
      =     "PL_Mov_Desc";
NETWORK
TITLE = Alarma en Almacenes
      O     "DB_OP".DF_003;
      O     "DB_OP".DF_095;
      O     "DB_OP".DF_103;
      O     "DB_OP".DF_002;
      =     "Alarma_Almacenes";
NETWORK
TITLE = Alarma en Araña
      O     "DB_OP".DF_004;
      O     "DB_OP".DF_065;
      O     "DB_OP".DF_066;
      O     "DB_OP".DF_067;
      O     "DB_OP".DF_068;
      O     "DB_OP".DF_073;
      O     "DB_OP".DF_074;
      =     "Alarma_Araña";
NETWORK
TITLE = Alarma en Rolos
      O     "DB_OP".DF_005;
      O     "DB_OP".DF_116;
      =     "Alarma_Rolos";
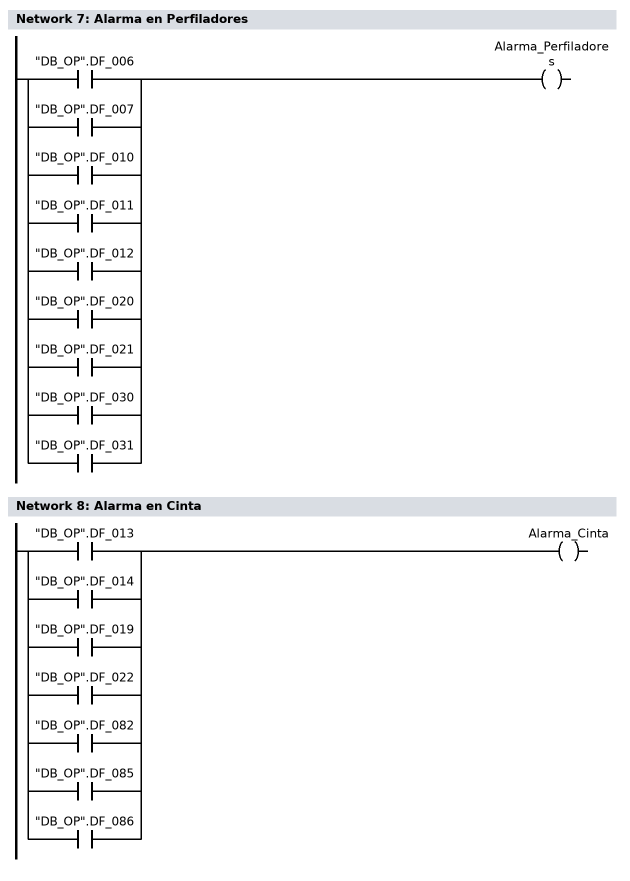
NETWORK
TITLE = Alarma en Perfiladores
      O     "DB_OP".DF_006;
      O     "DB_OP".DF_007;
      O     "DB_OP".DF_010;
      O     "DB_OP".DF_011;
      O     "DB_OP".DF_012;
      O     "DB_OP".DF_020;
      O     "DB_OP".DF_021;
      O     "DB_OP".DF_030;
      O     "DB_OP".DF_031;
      =     "Alarma_Perfiladores";
NETWORK
TITLE = Alarma en Cinta
      O     "DB_OP".DF_013;
      O     "DB_OP".DF_014;
      O     "DB_OP".DF_019;
      O     "DB_OP".DF_022;
      O     "DB_OP".DF_082;
      O     "DB_OP".DF_085;
      O     "DB_OP".DF_086;
      =     "Alarma_Cinta";
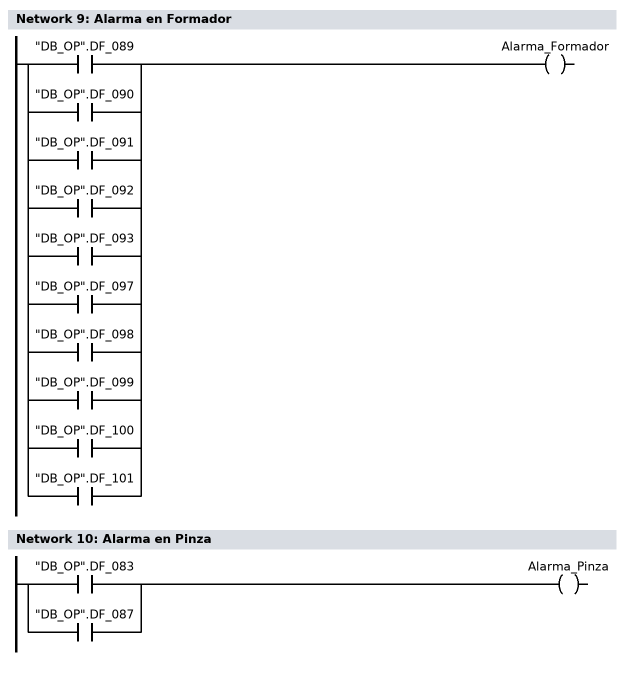
NETWORK
TITLE = Alarma en Formador
      O     "DB_OP".DF_089;
      O     "DB_OP".DF_090;
      O     "DB_OP".DF_091;
      O     "DB_OP".DF_092;
      O     "DB_OP".DF_093;
      O     "DB_OP".DF_097;
      O     "DB_OP".DF_098;
      O     "DB_OP".DF_099;
      O     "DB_OP".DF_100;
      O     "DB_OP".DF_101;
      =     "Alarma_Formador";
NETWORK
TITLE = Alarma en Pinza
      O     "DB_OP".DF_083;
      O     "DB_OP".DF_087;
      =     "Alarma_Pinza";
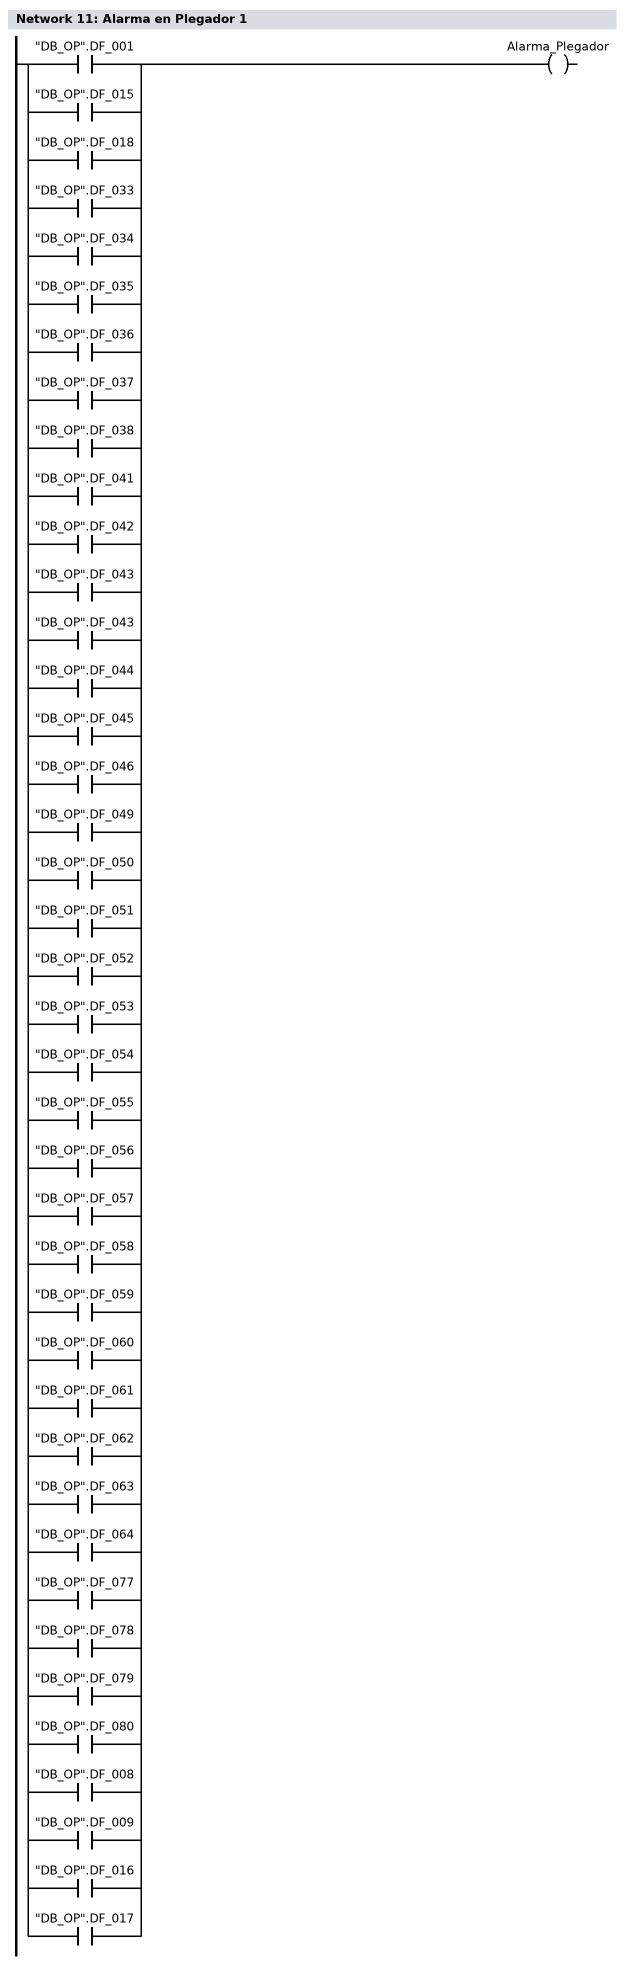
NETWORK
TITLE = Alarma en Plegador 1
      O     "DB_OP".DF_001;
      O     "DB_OP".DF_015;
      O     "DB_OP".DF_018;
      O     "DB_OP".DF_033;
      O     "DB_OP".DF_034;
      O     "DB_OP".DF_035;
      O     "DB_OP".DF_036;
      O     "DB_OP".DF_037;
      O     "DB_OP".DF_038;
      O     "DB_OP".DF_041;
      O     "DB_OP".DF_042;
      O     "DB_OP".DF_043;
      O     "DB_OP".DF_043;
      O     "DB_OP".DF_044;
      O     "DB_OP".DF_045;
      O     "DB_OP".DF_046;
      O     "DB_OP".DF_049;
      O     "DB_OP".DF_050;
      O     "DB_OP".DF_051;
      O     "DB_OP".DF_052;
      O     "DB_OP".DF_053;
      O     "DB_OP".DF_054;
      O     "DB_OP".DF_055;
      O     "DB_OP".DF_056;
      O     "DB_OP".DF_057;
      O     "DB_OP".DF_058;
      O     "DB_OP".DF_059;
      O     "DB_OP".DF_060;
      O     "DB_OP".DF_061;
      O     "DB_OP".DF_062;
      O     "DB_OP".DF_063;
      O     "DB_OP".DF_064;
      O     "DB_OP".DF_077;
      O     "DB_OP".DF_078;
      O     "DB_OP".DF_079;
      O     "DB_OP".DF_080;
      O     "DB_OP".DF_008;
      O     "DB_OP".DF_009;
      O     "DB_OP".DF_016;
      O     "DB_OP".DF_017;
      =     "Alarma_Plegador";
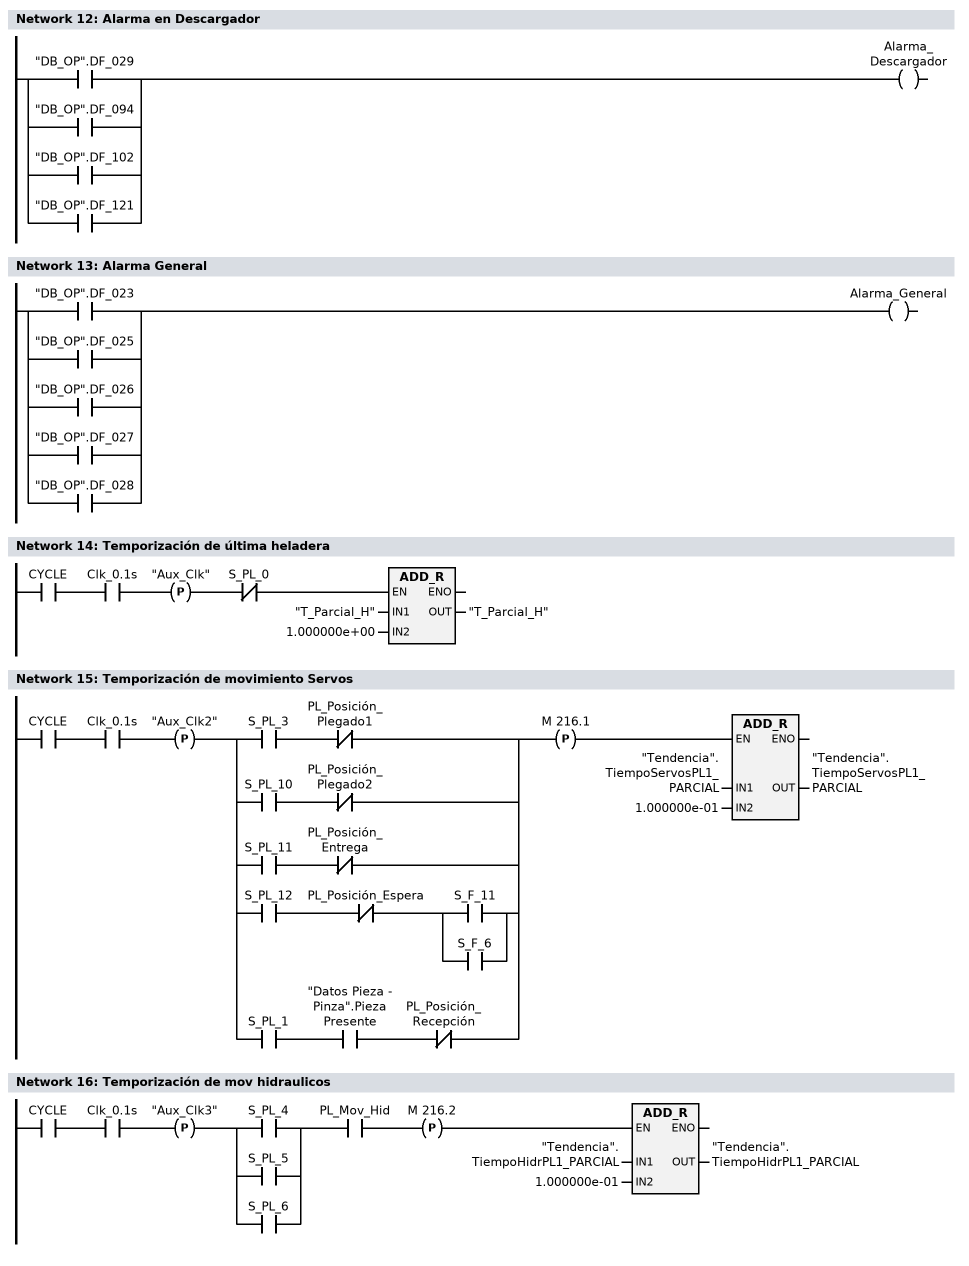
NETWORK
TITLE = Alarma en Descargador
      O     "DB_OP".DF_029;
      O     "DB_OP".DF_094;
      O     "DB_OP".DF_102;
      O     "DB_OP".DF_121;
      =     "Alarma_Descargador";
NETWORK
TITLE = Alarma General
      O     "DB_OP".DF_023;
      O     "DB_OP".DF_025;
      O     "DB_OP".DF_026;
      O     "DB_OP".DF_027;
      O     "DB_OP".DF_028;
      =     "Alarma_General";
NETWORK
TITLE = Temporización de última heladera
      A     "CYCLE";
      A(;
      A     "Clk_0.1s";
      BLD   100;
      FP    "Aux_Clk";
      );
      AN    "S_PL_0";
      JNB   _001;
      L     "T_Parcial_H";
      L     1.000000e+00;
      +R;
      T     "T_Parcial_H";
_001: NOP   0;
NETWORK
TITLE = Temporización de movimiento Servos
      A     "CYCLE";
      A(;
      A     "Clk_0.1s";
      BLD   100;
      FP    "Aux_Clk2";
      );
      A(;
      A     "S_PL_3";
      AN    "PL_Posición_Plegado1";
      O;
      A     "S_PL_10";
      AN    "PL_Posición_Plegado2";
      O;
      A     "S_PL_11";
      AN    "PL_Posición_Entrega";
      O;
      A     "S_PL_12";
      AN    "PL_Posición_Espera";
      A(;
      O     "S_F_11";
      O     "S_F_6";
      );
      O;
      A     "S_PL_1";
      A     "Datos Pieza - Pinza".PiezaPresente;
      AN    "PL_Posición_Recepción";
      );
      FP    M 216.1;
      JNB   _002;
      L     "Tendencia".TiempoServosPL1_PARCIAL;
      L     1.000000e-01;
      +R;
      T     "Tendencia".TiempoServosPL1_PARCIAL;
_002: NOP   0;
NETWORK
TITLE = Temporización de mov hidraulicos
      A     "CYCLE";
      A(;
      A     "Clk_0.1s";
      BLD   100;
      FP    "Aux_Clk3";
      );
      A(;
      O     "S_PL_4";
      O     "S_PL_5";
      O     "S_PL_6";
      );
      A     "PL_Mov_Hid";
      FP    M 216.2;
      JNB   _003;
      L     "Tendencia".TiempoHidrPL1_PARCIAL;
      L     1.000000e-01;
      +R;
      T     "Tendencia".TiempoHidrPL1_PARCIAL;
_003: NOP   0;
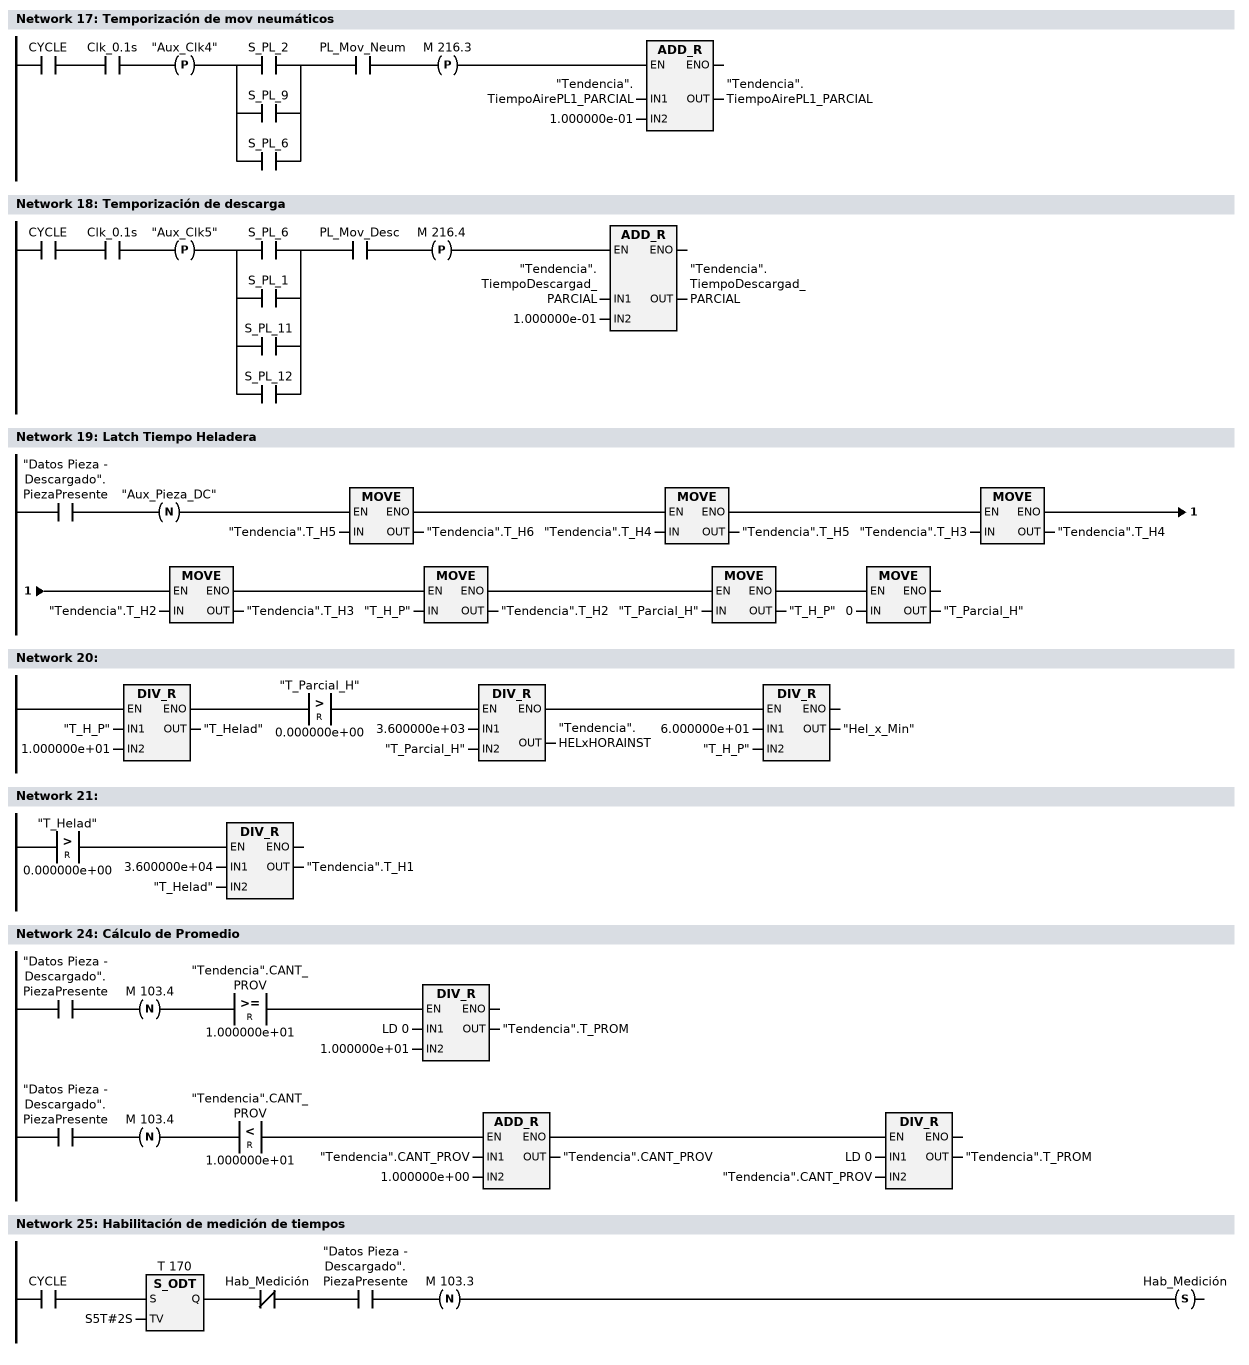
NETWORK
TITLE = Temporización de mov neumáticos
      A     "CYCLE";
      A(;
      A     "Clk_0.1s";
      BLD   100;
      FP    "Aux_Clk4";
      );
      A(;
      O     "S_PL_2";
      O     "S_PL_9";
      O     "S_PL_6";
      );
      A     "PL_Mov_Neum";
      FP    M 216.3;
      JNB   _004;
      L     "Tendencia".TiempoAirePL1_PARCIAL;
      L     1.000000e-01;
      +R;
      T     "Tendencia".TiempoAirePL1_PARCIAL;
_004: NOP   0;
NETWORK
TITLE = Temporización de descarga
      A     "CYCLE";
      A(;
      A     "Clk_0.1s";
      BLD   100;
      FP    "Aux_Clk5";
      );
      A(;
      O     "S_PL_6";
      O     "S_PL_1";
      O     "S_PL_11";
      O     "S_PL_12";
      );
      A     "PL_Mov_Desc";
      FP    M 216.4;
      JNB   _005;
      L     "Tendencia".TiempoDescargad_PARCIAL;
      L     1.000000e-01;
      +R;
      T     "Tendencia".TiempoDescargad_PARCIAL;
_005: NOP   0;
NETWORK
TITLE = Latch Tiempo Heladera
      A(;
      A(;
      A(;
      A(;
      A(;
      A(;
      A     "Datos Pieza - Descargado".PiezaPresente;
      FN    "Aux_Pieza_DC";
      JNB   _006;
      L     "Tendencia".T_H5;
      T     "Tendencia".T_H6;
      SET;
      SAVE;
      CLR;
_006: A     BR;
      );
      JNB   _007;
      L     "Tendencia".T_H4;
      T     "Tendencia".T_H5;
      SET;
      SAVE;
      CLR;
_007: A     BR;
      );
      JNB   _008;
      L     "Tendencia".T_H3;
      T     "Tendencia".T_H4;
      SET;
      SAVE;
      CLR;
_008: A     BR;
      );
      JNB   _009;
      L     "Tendencia".T_H2;
      T     "Tendencia".T_H3;
      SET;
      SAVE;
      CLR;
_009: A     BR;
      );
      JNB   _00a;
      L     "T_H_P";
      T     "Tendencia".T_H2;
      SET;
      SAVE;
      CLR;
_00a: A     BR;
      );
      JNB   _00b;
      L     "T_Parcial_H";
      T     "T_H_P";
      SET;
      SAVE;
      CLR;
_00b: A     BR;
      );
      JNB   _00c;
      L     0;
      T     "T_Parcial_H";
_00c: NOP   0;
NETWORK
TITLE =
      A(;
      A(;
      L     "T_H_P";
      L     1.000000e+01;
      /R;
      T     "T_Helad";
      AN    OV;
      SAVE;
      CLR;
      A     BR;
      );
      A(;
      L     "T_Parcial_H";
      L     0.000000e+00;
      >R;
      );
      JNB   _00d;
      L     3.600000e+03;
      L     "T_Parcial_H";
      /R;
      T     "Tendencia".HELxHORAINST;
      AN    OV;
      SAVE;
      CLR;
_00d: A     BR;
      );
      JNB   _00e;
      L     6.000000e+01;
      L     "T_H_P";
      /R;
      T     "Hel_x_Min";
_00e: NOP   0;
NETWORK
TITLE =
      A(;
      L     "T_Helad";
      L     0.000000e+00;
      >R;
      );
      JNB   _00f;
      L     3.600000e+04;
      L     "T_Helad";
      /R;
      T     "Tendencia".T_H1;
_00f: NOP   0;
NETWORK
TITLE = Suma Total de Tiempos
      L     "Tendencia".T_H1;
      L     "Tendencia".T_H2;
      +R;
      L     "Tendencia".T_H3;
      +R;
      L     "Tendencia".T_H4;
      +R;
      L     "Tendencia".T_H5;
      +R;
      L     "Tendencia".T_H6;
      +R;
      L     "Tendencia".T_H7;
      +R;
      L     "Tendencia".T_H8;
      +R;
      L     "Tendencia".T_H9;
      +R;
      L     "Tendencia".T_H10;
      +R;
      T     LD 0;
NETWORK
TITLE = Reseteo de Valores por máquina fuera de ciclo
      A     "CYCLE";
      JC    M013;
      L     0.000000e+00;
//    T     "Tendencia".T_H1
//    T    "Tendencia".T_H2
//    T     "Tendencia".T_H3
//    T     "Tendencia".T_H4
//    T     "Tendencia".T_H5
//    T     "Tendencia".T_H6
//    T     "Tendencia".T_H7
//    T     "Tendencia".T_H8
//    T     "Tendencia".T_H9
//    T     "Tendencia".T_H10
//    T     "Tendencia".CANT_PROV
//    T     "Tendencia".T_PROM
//    T     "Hel_x_Min"
//    T     "Hel_x_H"
//    T     "T_Helad"
M013: NOP   0;
NETWORK
TITLE = Cálculo de Promedio
      A     "Datos Pieza - Descargado".PiezaPresente;
      FN    M 103.4;
      =     L 4.0;
      A(;
      A     L 4.0;
      A(;
      L     "Tendencia".CANT_PROV;
      L     1.000000e+01;
      <R;
      );
      JNB   _010;
      L     "Tendencia".CANT_PROV;
      L     1.000000e+00;
      +R;
      T     "Tendencia".CANT_PROV;
      AN    OV;
      SAVE;
      CLR;
_010: A     BR;
      );
      JNB   _011;
      L     LD 0;
      L     "Tendencia".CANT_PROV;
      /R;
      T     "Tendencia".T_PROM;
_011: NOP   0;
      A     L 4.0;
      A(;
      L     "Tendencia".CANT_PROV;
      L     1.000000e+01;
      >=R;
      );
      JNB   _012;
      L     LD 0;
      L     1.000000e+01;
      /R;
      T     "Tendencia".T_PROM;
_012: NOP   0;
NETWORK
TITLE = Habilitación de medición de tiempos
      A(;
      A     "CYCLE";
      L     S5T#2S;
      SD    T 170;
      NOP   0;
      NOP   0;
      NOP   0;
      A     T 170;
      );
      AN    "Hab_Medición";
      A(;
      A     "Datos Pieza - Descargado".PiezaPresente;
      BLD   100;
      FN    M 103.3;
      );
      S     "Hab_Medición";
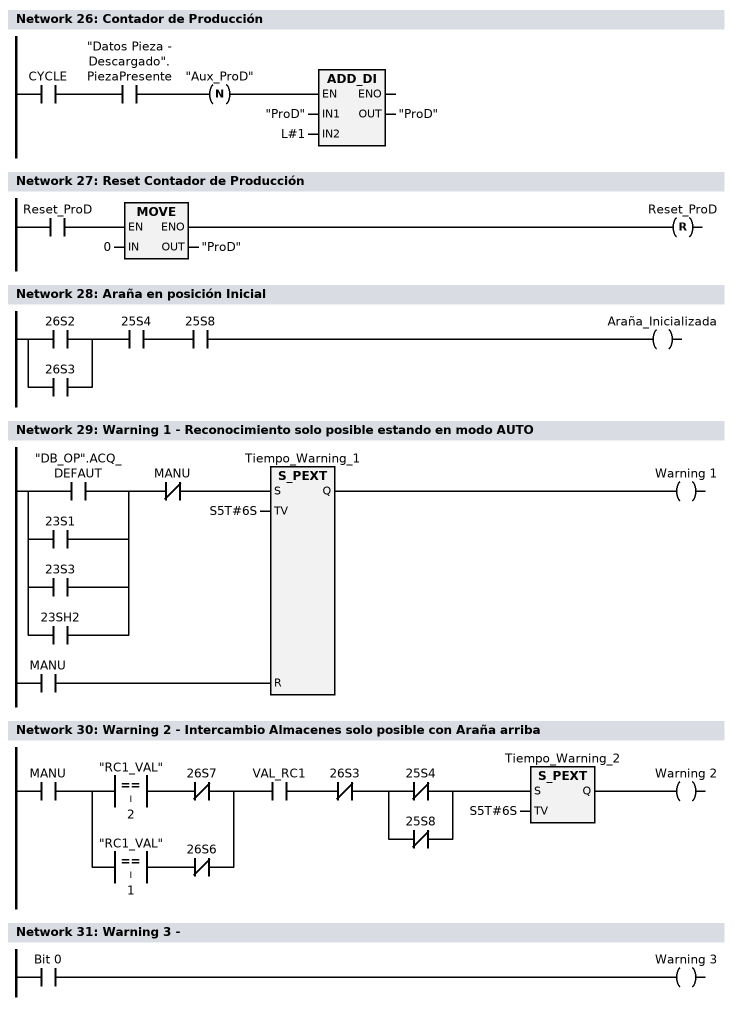
NETWORK
TITLE = Contador de Producción
      A     "CYCLE";
      A(;
      A     "Datos Pieza - Descargado".PiezaPresente;
      BLD   100;
      FN    "Aux_ProD";
      );
      JNB   _013;
      L     "ProD";
      L     L#1;
      +D;
      T     "ProD";
_013: NOP   0;
NETWORK
TITLE = Reset Contador de Producción
      A     "Reset_ProD";
      JNB   _014;
      L     0;
      T     "ProD";
      SET;
      SAVE;
      CLR;
_014: A     BR;
      R     "Reset_ProD";
NETWORK
TITLE = Araña en posición Inicial
      A(;
      O     "26S2";
      O     "26S3";
      );
      A     "25S4";
      A     "25S8";
      =     "Araña_Inicializada";
NETWORK
TITLE = Warning 1 - Reconocimiento solo posible estando en modo AUTO
      A(;
      O     "DB_OP".ACQ_DEFAUT;
      O     "23S1";
      O     "23S3";
      O     "23SH2";
      );
      AN    "MANU";
      L     S5T#6S;
      SE    "Tiempo_Warning_1";
      A     "MANU";
      R     "Tiempo_Warning_1";
      NOP   0;
      NOP   0;
      A     "Tiempo_Warning_1";
      =     "Warning 1";
NETWORK
TITLE = Warning 2 - Intercambio Almacenes solo posible con Araña arriba
      A     "MANU";
      A(;
      A(;
      L     "RC1_VAL";
      L     2;
      ==I;
      );
      AN    "26S7";
      O;
      A(;
      L     "RC1_VAL";
      L     1;
      ==I;
      );
      AN    "26S6";
      );
      A     "VAL_RC1";
      AN    "26S3";
      A(;
      ON    "25S4";
      ON    "25S8";
      );
      L     S5T#6S;
      SE    "Tiempo_Warning_2";
      NOP   0;
      NOP   0;
      NOP   0;
      A     "Tiempo_Warning_2";
      =     "Warning 2";
NETWORK
TITLE = Warning 3 -
      A     "Bit 0";
      =     "Warning 3";
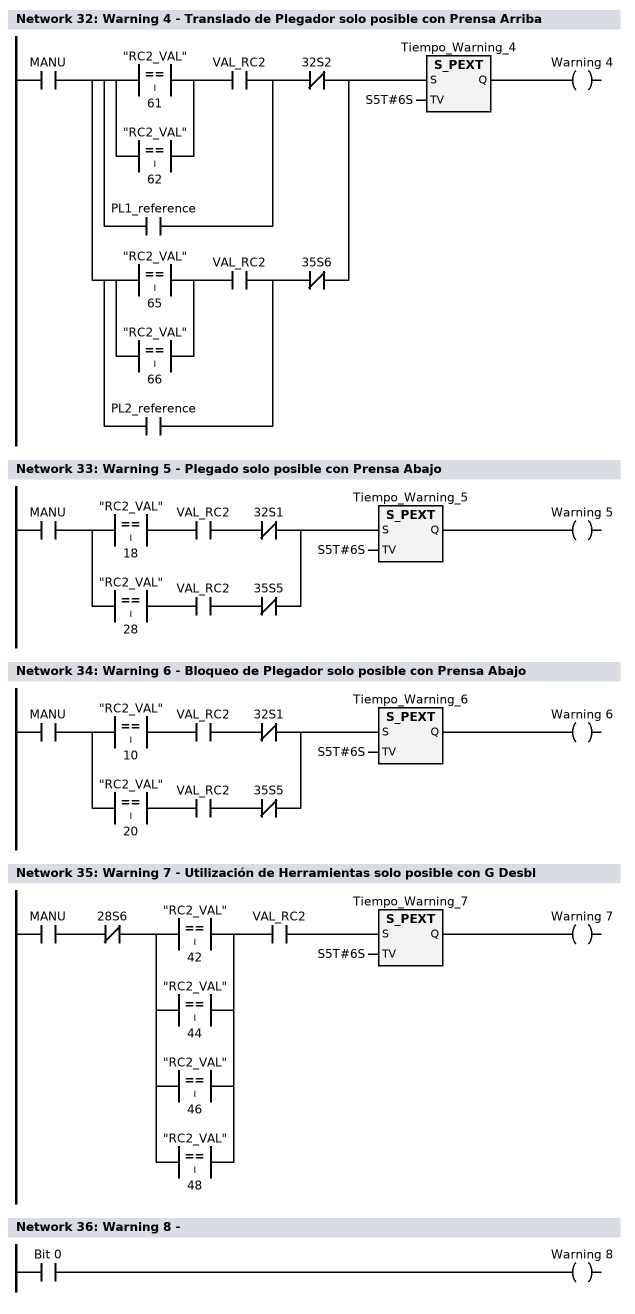
NETWORK
TITLE = Warning 4 - Translado de Plegador solo posible con Prensa Arriba
      A     "MANU";
      A(;
      A(;
      A(;
      O(;
      L     "RC2_VAL";
      L     61;
      ==I;
      );
      O(;
      L     "RC2_VAL";
      L     62;
      ==I;
      );
      );
      A     "VAL_RC2";
      O     "PL1_reference";
      );
      AN    "32S2";
      O;
      A(;
      A(;
      O(;
      L     "RC2_VAL";
      L     65;
      ==I;
      );
      O(;
      L     "RC2_VAL";
      L     66;
      ==I;
      );
      );
      A     "VAL_RC2";
      O     "PL2_reference";
      );
      AN    "35S6";
      );
      L     S5T#6S;
      SE    "Tiempo_Warning_4";
      NOP   0;
      NOP   0;
      NOP   0;
      A     "Tiempo_Warning_4";
      =     "Warning 4";
NETWORK
TITLE = Warning 5 - Plegado solo posible con Prensa Abajo
      A     "MANU";
      A(;
      A(;
      L     "RC2_VAL";
      L     18;
      ==I;
      );
      A     "VAL_RC2";
      AN    "32S1";
      O;
      A(;
      L     "RC2_VAL";
      L     28;
      ==I;
      );
      A     "VAL_RC2";
      AN    "35S5";
      );
      L     S5T#6S;
      SE    "Tiempo_Warning_5";
      NOP   0;
      NOP   0;
      NOP   0;
      A     "Tiempo_Warning_5";
      =     "Warning 5";
NETWORK
TITLE = Warning 6 - Bloqueo de Plegador solo posible con Prensa Abajo
      A     "MANU";
      A(;
      A(;
      L     "RC2_VAL";
      L     10;
      ==I;
      );
      A     "VAL_RC2";
      AN    "32S1";
      O;
      A(;
      L     "RC2_VAL";
      L     20;
      ==I;
      );
      A     "VAL_RC2";
      AN    "35S5";
      );
      L     S5T#6S;
      SE    "Tiempo_Warning_6";
      NOP   0;
      NOP   0;
      NOP   0;
      A     "Tiempo_Warning_6";
      =     "Warning 6";
NETWORK
TITLE = Warning 7 - Utilización de Herramientas solo posible con G Desbl
      A     "MANU";
      AN    "28S6";
      A(;
      O(;
      L     "RC2_VAL";
      L     42;
      ==I;
      );
      O(;
      L     "RC2_VAL";
      L     44;
      ==I;
      );
      O(;
      L     "RC2_VAL";
      L     46;
      ==I;
      );
      O(;
      L     "RC2_VAL";
      L     48;
      ==I;
      );
      );
      A     "VAL_RC2";
      L     S5T#6S;
      SE    "Tiempo_Warning_7";
      NOP   0;
      NOP   0;
      NOP   0;
      A     "Tiempo_Warning_7";
      =     "Warning 7";
NETWORK
TITLE = Warning 8 - 
      A     "Bit 0";
      =     "Warning 8";
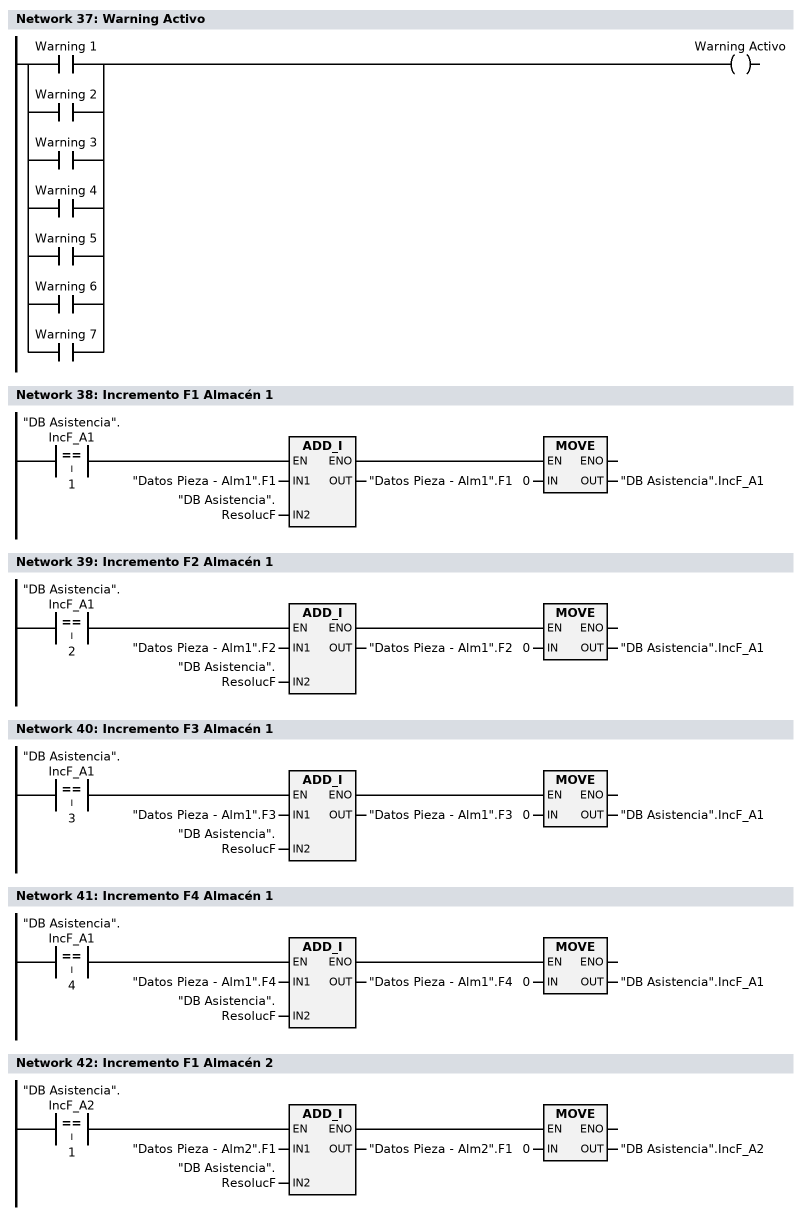
NETWORK
TITLE = Warning Activo
      O     "Warning 1";
      O     "Warning 2";
      O     "Warning 3";
      O     "Warning 4";
      O     "Warning 5";
      O     "Warning 6";
      O     "Warning 7";
      =     "Warning Activo";
NETWORK
TITLE = Incremento F1 Almacén 1
      A(;
      A(;
      L     "DB Asistencia".IncF_A1;
      L     1;
      ==I;
      );
      JNB   _015;
      L     "Datos Pieza - Alm1".F1;
      L     "DB Asistencia".ResolucF;
      +I;
      T     "Datos Pieza - Alm1".F1;
      AN    OV;
      SAVE;
      CLR;
_015: A     BR;
      );
      JNB   _016;
      L     0;
      T     "DB Asistencia".IncF_A1;
_016: NOP   0;
NETWORK
TITLE = Incremento F2 Almacén 1
      A(;
      A(;
      L     "DB Asistencia".IncF_A1;
      L     2;
      ==I;
      );
      JNB   _017;
      L     "Datos Pieza - Alm1".F2;
      L     "DB Asistencia".ResolucF;
      +I;
      T     "Datos Pieza - Alm1".F2;
      AN    OV;
      SAVE;
      CLR;
_017: A     BR;
      );
      JNB   _018;
      L     0;
      T     "DB Asistencia".IncF_A1;
_018: NOP   0;
NETWORK
TITLE = Incremento F3 Almacén 1
      A(;
      A(;
      L     "DB Asistencia".IncF_A1;
      L     3;
      ==I;
      );
      JNB   _019;
      L     "Datos Pieza - Alm1".F3;
      L     "DB Asistencia".ResolucF;
      +I;
      T     "Datos Pieza - Alm1".F3;
      AN    OV;
      SAVE;
      CLR;
_019: A     BR;
      );
      JNB   _01a;
      L     0;
      T     "DB Asistencia".IncF_A1;
_01a: NOP   0;
NETWORK
TITLE = Incremento F4 Almacén 1
      A(;
      A(;
      L     "DB Asistencia".IncF_A1;
      L     4;
      ==I;
      );
      JNB   _01b;
      L     "Datos Pieza - Alm1".F4;
      L     "DB Asistencia".ResolucF;
      +I;
      T     "Datos Pieza - Alm1".F4;
      AN    OV;
      SAVE;
      CLR;
_01b: A     BR;
      );
      JNB   _01c;
      L     0;
      T     "DB Asistencia".IncF_A1;
_01c: NOP   0;
NETWORK
TITLE = Incremento F1 Almacén 2
      A(;
      A(;
      L     "DB Asistencia".IncF_A2;
      L     1;
      ==I;
      );
      JNB   _01d;
      L     "Datos Pieza - Alm2".F1;
      L     "DB Asistencia".ResolucF;
      +I;
      T     "Datos Pieza - Alm2".F1;
      AN    OV;
      SAVE;
      CLR;
_01d: A     BR;
      );
      JNB   _01e;
      L     0;
      T     "DB Asistencia".IncF_A2;
_01e: NOP   0;
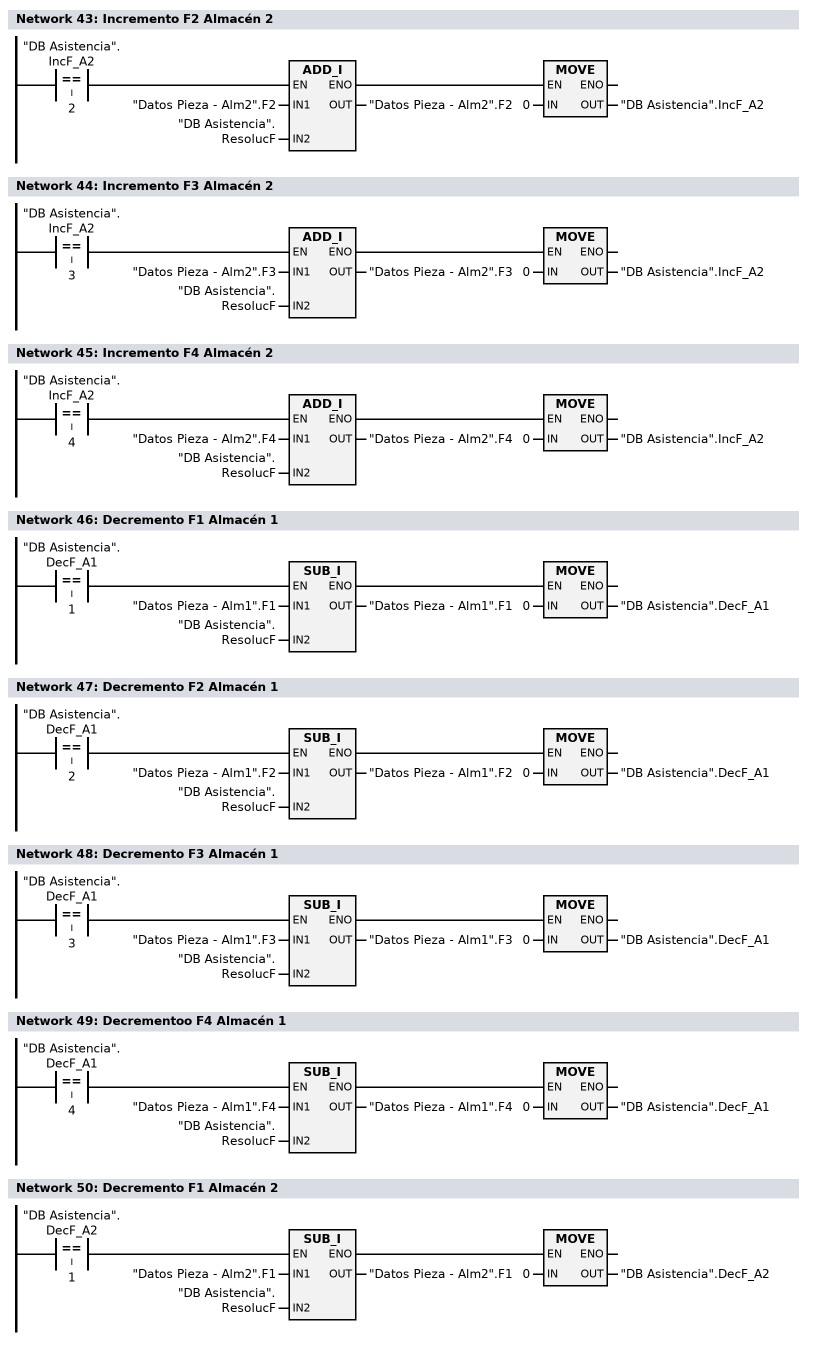
NETWORK
TITLE = Incremento F2 Almacén 2
      A(;
      A(;
      L     "DB Asistencia".IncF_A2;
      L     2;
      ==I;
      );
      JNB   _01f;
      L     "Datos Pieza - Alm2".F2;
      L     "DB Asistencia".ResolucF;
      +I;
      T     "Datos Pieza - Alm2".F2;
      AN    OV;
      SAVE;
      CLR;
_01f: A     BR;
      );
      JNB   _020;
      L     0;
      T     "DB Asistencia".IncF_A2;
_020: NOP   0;
NETWORK
TITLE = Incremento F3 Almacén 2
      A(;
      A(;
      L     "DB Asistencia".IncF_A2;
      L     3;
      ==I;
      );
      JNB   _021;
      L     "Datos Pieza - Alm2".F3;
      L     "DB Asistencia".ResolucF;
      +I;
      T     "Datos Pieza - Alm2".F3;
      AN    OV;
      SAVE;
      CLR;
_021: A     BR;
      );
      JNB   _022;
      L     0;
      T     "DB Asistencia".IncF_A2;
_022: NOP   0;
NETWORK
TITLE = Incremento F4 Almacén 2
      A(;
      A(;
      L     "DB Asistencia".IncF_A2;
      L     4;
      ==I;
      );
      JNB   _023;
      L     "Datos Pieza - Alm2".F4;
      L     "DB Asistencia".ResolucF;
      +I;
      T     "Datos Pieza - Alm2".F4;
      AN    OV;
      SAVE;
      CLR;
_023: A     BR;
      );
      JNB   _024;
      L     0;
      T     "DB Asistencia".IncF_A2;
_024: NOP   0;
NETWORK
TITLE = Decremento F1 Almacén 1
      A(;
      A(;
      L     "DB Asistencia".DecF_A1;
      L     1;
      ==I;
      );
      JNB   _025;
      L     "Datos Pieza - Alm1".F1;
      L     "DB Asistencia".ResolucF;
      -I;
      T     "Datos Pieza - Alm1".F1;
      AN    OV;
      SAVE;
      CLR;
_025: A     BR;
      );
      JNB   _026;
      L     0;
      T     "DB Asistencia".DecF_A1;
_026: NOP   0;
NETWORK
TITLE = Decremento F2 Almacén 1
      A(;
      A(;
      L     "DB Asistencia".DecF_A1;
      L     2;
      ==I;
      );
      JNB   _027;
      L     "Datos Pieza - Alm1".F2;
      L     "DB Asistencia".ResolucF;
      -I;
      T     "Datos Pieza - Alm1".F2;
      AN    OV;
      SAVE;
      CLR;
_027: A     BR;
      );
      JNB   _028;
      L     0;
      T     "DB Asistencia".DecF_A1;
_028: NOP   0;
NETWORK
TITLE = Decremento F3 Almacén 1
      A(;
      A(;
      L     "DB Asistencia".DecF_A1;
      L     3;
      ==I;
      );
      JNB   _029;
      L     "Datos Pieza - Alm1".F3;
      L     "DB Asistencia".ResolucF;
      -I;
      T     "Datos Pieza - Alm1".F3;
      AN    OV;
      SAVE;
      CLR;
_029: A     BR;
      );
      JNB   _02a;
      L     0;
      T     "DB Asistencia".DecF_A1;
_02a: NOP   0;
NETWORK
TITLE = Decrementoo F4 Almacén 1
      A(;
      A(;
      L     "DB Asistencia".DecF_A1;
      L     4;
      ==I;
      );
      JNB   _02b;
      L     "Datos Pieza - Alm1".F4;
      L     "DB Asistencia".ResolucF;
      -I;
      T     "Datos Pieza - Alm1".F4;
      AN    OV;
      SAVE;
      CLR;
_02b: A     BR;
      );
      JNB   _02c;
      L     0;
      T     "DB Asistencia".DecF_A1;
_02c: NOP   0;
NETWORK
TITLE = Decremento F1 Almacén 2
      A(;
      A(;
      L     "DB Asistencia".DecF_A2;
      L     1;
      ==I;
      );
      JNB   _02d;
      L     "Datos Pieza - Alm2".F1;
      L     "DB Asistencia".ResolucF;
      -I;
      T     "Datos Pieza - Alm2".F1;
      AN    OV;
      SAVE;
      CLR;
_02d: A     BR;
      );
      JNB   _02e;
      L     0;
      T     "DB Asistencia".DecF_A2;
_02e: NOP   0;
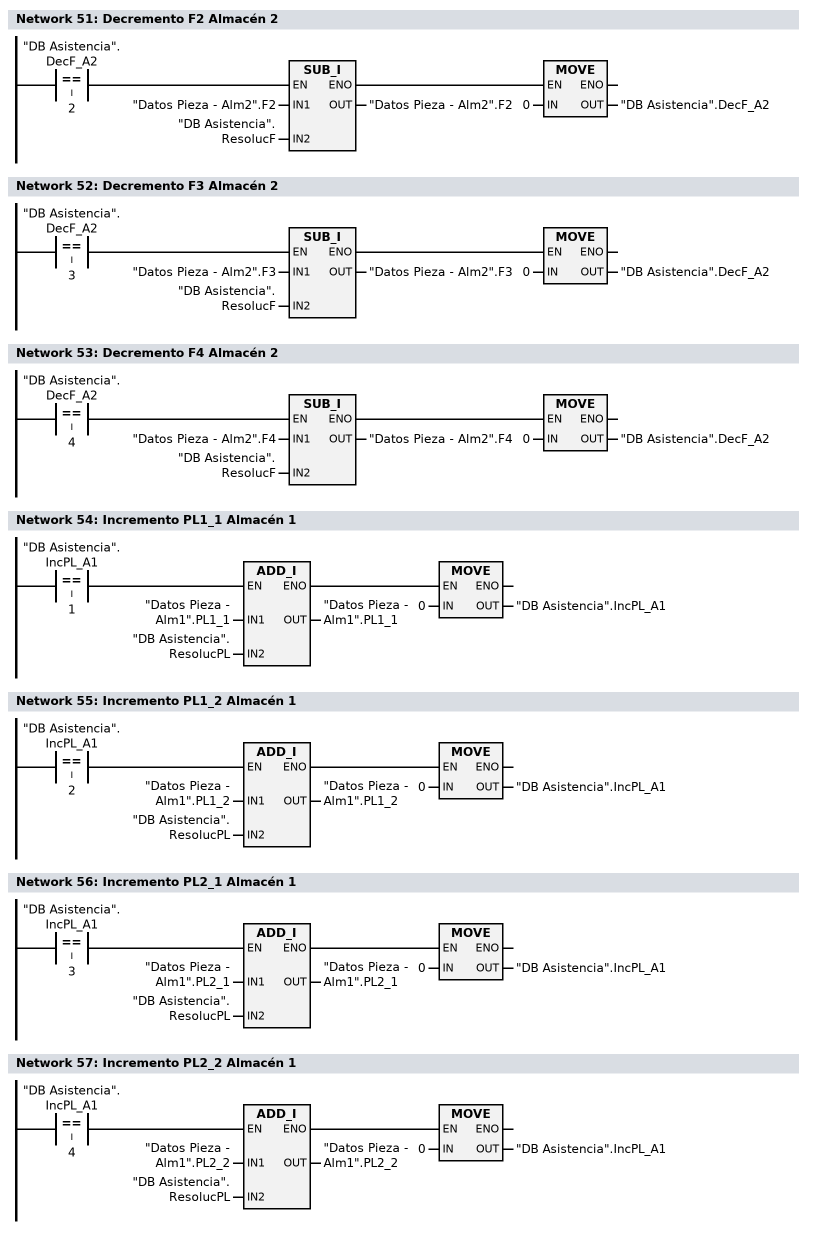
NETWORK
TITLE = Decremento F2 Almacén 2
      A(;
      A(;
      L     "DB Asistencia".DecF_A2;
      L     2;
      ==I;
      );
      JNB   _02f;
      L     "Datos Pieza - Alm2".F2;
      L     "DB Asistencia".ResolucF;
      -I;
      T     "Datos Pieza - Alm2".F2;
      AN    OV;
      SAVE;
      CLR;
_02f: A     BR;
      );
      JNB   _030;
      L     0;
      T     "DB Asistencia".DecF_A2;
_030: NOP   0;
NETWORK
TITLE = Decremento F3 Almacén 2
      A(;
      A(;
      L     "DB Asistencia".DecF_A2;
      L     3;
      ==I;
      );
      JNB   _031;
      L     "Datos Pieza - Alm2".F3;
      L     "DB Asistencia".ResolucF;
      -I;
      T     "Datos Pieza - Alm2".F3;
      AN    OV;
      SAVE;
      CLR;
_031: A     BR;
      );
      JNB   _032;
      L     0;
      T     "DB Asistencia".DecF_A2;
_032: NOP   0;
NETWORK
TITLE = Decremento F4 Almacén 2
      A(;
      A(;
      L     "DB Asistencia".DecF_A2;
      L     4;
      ==I;
      );
      JNB   _033;
      L     "Datos Pieza - Alm2".F4;
      L     "DB Asistencia".ResolucF;
      -I;
      T     "Datos Pieza - Alm2".F4;
      AN    OV;
      SAVE;
      CLR;
_033: A     BR;
      );
      JNB   _034;
      L     0;
      T     "DB Asistencia".DecF_A2;
_034: NOP   0;
NETWORK
TITLE = Incremento PL1_1 Almacén 1
      A(;
      A(;
      L     "DB Asistencia".IncPL_A1;
      L     1;
      ==I;
      );
      JNB   _035;
      L     "Datos Pieza - Alm1".PL1_1;
      L     "DB Asistencia".ResolucPL;
      +I;
      T     "Datos Pieza - Alm1".PL1_1;
      AN    OV;
      SAVE;
      CLR;
_035: A     BR;
      );
      JNB   _036;
      L     0;
      T     "DB Asistencia".IncPL_A1;
_036: NOP   0;
NETWORK
TITLE = Incremento PL1_2 Almacén 1
      A(;
      A(;
      L     "DB Asistencia".IncPL_A1;
      L     2;
      ==I;
      );
      JNB   _037;
      L     "Datos Pieza - Alm1".PL1_2;
      L     "DB Asistencia".ResolucPL;
      +I;
      T     "Datos Pieza - Alm1".PL1_2;
      AN    OV;
      SAVE;
      CLR;
_037: A     BR;
      );
      JNB   _038;
      L     0;
      T     "DB Asistencia".IncPL_A1;
_038: NOP   0;
NETWORK
TITLE = Incremento PL2_1 Almacén 1
      A(;
      A(;
      L     "DB Asistencia".IncPL_A1;
      L     3;
      ==I;
      );
      JNB   _039;
      L     "Datos Pieza - Alm1".PL2_1;
      L     "DB Asistencia".ResolucPL;
      +I;
      T     "Datos Pieza - Alm1".PL2_1;
      AN    OV;
      SAVE;
      CLR;
_039: A     BR;
      );
      JNB   _03a;
      L     0;
      T     "DB Asistencia".IncPL_A1;
_03a: NOP   0;
NETWORK
TITLE = Incremento PL2_2 Almacén 1
      A(;
      A(;
      L     "DB Asistencia".IncPL_A1;
      L     4;
      ==I;
      );
      JNB   _03b;
      L     "Datos Pieza - Alm1".PL2_2;
      L     "DB Asistencia".ResolucPL;
      +I;
      T     "Datos Pieza - Alm1".PL2_2;
      AN    OV;
      SAVE;
      CLR;
_03b: A     BR;
      );
      JNB   _03c;
      L     0;
      T     "DB Asistencia".IncPL_A1;
_03c: NOP   0;
